C08983=1030.754,339.492,-131.948,171.836,46.140,159.013
C08984=1030.746,339.245,-131.912,171.829,46.139,159.012
C08985=1030.738,338.997,-131.876,171.824,46.139,159.011
C08986=1030.731,338.751,-131.839,171.818,46.137,159.010
C08987=1030.723,338.504,-131.803,171.812,46.137,159.009
C08988=1030.716,338.256,-131.767,171.806,46.135,159.008
C08989=1030.709,338.008,-131.730,171.800,46.135,159.007
C08990=1030.701,337.761,-131.694,171.795,46.133,159.006
C08991=1030.694,337.514,-131.658,171.789,46.133,159.006
C08992=1030.686,337.267,-131.621,171.783,46.132,159.005
C08993=1030.678,337.020,-131.585,171.778,46.131,159.004
C08994=1030.671,336.772,-131.549,171.772,46.130,159.003
C08995=1030.663,336.526,-131.513,171.766,46.129,159.002
C08996=1030.651,336.113,-131.452,171.757,46.128,159.001
C08997=1030.639,335.700,-131.391,171.748,46.126,158.999
C08998=1030.627,335.287,-131.331,171.738,46.124,158.998
C08999=1030.615,334.875,-131.271,171.729,46.123,158.996
C09000=1030.607,334.627,-131.235,171.723,46.123,158.996
C09001=1030.600,334.381,-131.199,171.718,46.121,158.995
C09002=1030.592,334.133,-131.163,171.712,46.121,158.994
C09003=1030.585,333.886,-131.128,171.707,46.120,158.993
C09004=1030.578,333.638,-131.091,171.701,46.119,158.992
C09005=1030.570,333.391,-131.055,171.695,46.119,158.991
C09006=1030.563,333.143,-131.020,171.690,46.118,158.991
C09007=1030.555,332.896,-130.984,171.684,46.117,158.990
C09008=1030.547,332.649,-130.948,171.678,46.117,158.989
C09009=1030.540,332.402,-130.913,171.673,46.116,158.988
C09010=1030.533,332.154,-130.877,171.667,46.115,158.987
C09011=1030.526,331.907,-130.841,171.662,46.114,158.987
C09012=1030.518,331.659,-130.806,171.656,46.113,158.986
C09013=1030.511,331.413,-130.770,171.651,46.113,158.985
C09014=1030.504,331.164,-130.734,171.646,46.112,158.984
C09015=1030.497,330.918,-130.698,171.640,46.111,158.983
C09016=1030.489,330.670,-130.663,171.635,46.111,158.983
C09017=1030.482,330.423,-130.628,171.629,46.111,158.982
C09018=1030.474,330.175,-130.592,171.624,46.110,158.981
C09019=1030.467,329.928,-130.556,171.619,46.109,158.980
C09020=1030.460,329.680,-130.521,171.613,46.109,158.980
C09021=1030.453,329.434,-130.485,171.608,46.108,158.979
C09022=1030.445,329.186,-130.449,171.602,46.107,158.978
C09023=1030.438,328.938,-130.415,171.597,46.106,158.977
C09024=1030.431,328.692,-130.379,171.591,46.106,158.976
C09025=1030.423,328.444,-130.343,171.586,46.105,158.976
C09026=1030.417,328.196,-130.308,171.581,46.105,158.975
C09027=1030.409,327.949,-130.272,171.576,46.104,158.974
C09028=1030.402,327.702,-130.237,171.570,46.104,158.974
C09029=1030.395,327.454,-130.202,171.565,46.103,158.973
C09030=1030.387,327.207,-130.168,171.559,46.103,158.972
C09031=1030.380,326.959,-130.132,171.554,46.102,158.971
C09032=1030.372,326.712,-130.098,171.548,46.101,158.971
C09033=1030.365,326.464,-130.062,171.543,46.101,158.970
C09034=1030.357,326.217,-130.028,171.538,46.101,158.969
C09035=1030.350,325.970,-129.992,171.532,46.101,158.969
C09036=1030.342,325.723,-129.957,171.528,46.100,158.968
C09037=1030.336,325.475,-129.923,171.522,46.100,158.967
C09038=1030.328,325.227,-129.888,171.517,46.099,158.966
C09039=1030.320,324.980,-129.853,171.511,46.098,158.966
C09040=1030.313,324.733,-129.818,171.507,46.098,158.965
C09041=1030.305,324.485,-129.783,171.501,46.098,158.964
C09042=1030.299,324.237,-129.748,171.496,46.097,158.964
C09043=1030.291,323.990,-129.714,171.490,46.097,158.963
C09044=1030.284,323.742,-129.678,171.486,46.097,158.962
C09045=1030.276,323.495,-129.643,171.480,46.097,158.962
C09046=1030.269,323.248,-129.609,171.475,46.096,158.961
C09047=1030.262,323.000,-129.575,171.469,46.096,158.960
C09048=1030.254,322.752,-129.540,171.465,46.095,158.959
C09049=1030.247,322.505,-129.504,171.459,46.095,158.959
C09050=1030.240,322.258,-129.470,171.454,46.095,158.958
C09051=1030.233,322.010,-129.436,171.449,46.094,158.957
C09052=1030.221,321.593,-129.377,171.440,46.093,158.956
C09053=1030.208,321.176,-129.319,171.432,46.093,158.955
C09054=1030.196,320.759,-129.260,171.423,46.092,158.954
C09055=1030.184,320.342,-129.203,171.415,46.092,158.953
C09056=1030.178,320.095,-129.167,171.409,46.092,158.952
C09057=1030.170,319.848,-129.133,171.404,46.091,158.952
C09058=1030.162,319.599,-129.099,171.400,46.091,158.951
C09059=1030.156,319.352,-129.064,171.394,46.091,158.950
C09060=1030.148,319.104,-129.030,171.389,46.090,158.950
C09061=1030.142,318.857,-128.995,171.384,46.090,158.949
C09062=1030.134,318.609,-128.961,171.379,46.090,158.949
C09063=1030.127,318.362,-128.926,171.374,46.089,158.948
C09064=1030.120,318.114,-128.892,171.369,46.089,158.947
C09065=1030.113,317.867,-128.857,171.364,46.089,158.947
C09066=1030.106,317.619,-128.824,171.359,46.089,158.946
C09067=1030.099,317.372,-128.788,171.354,46.089,158.945
C09068=1030.092,317.124,-128.755,171.349,46.089,158.945
C09069=1030.085,316.876,-128.720,171.344,46.089,158.944
C09070=1030.078,316.629,-128.686,171.339,46.088,158.943
C09071=1030.071,316.382,-128.652,171.334,46.088,158.943
C09072=1030.064,316.134,-128.617,171.329,46.088,158.942
C09073=1030.057,315.887,-128.583,171.324,46.087,158.942
C09074=1030.050,315.640,-128.549,171.319,46.087,158.941
C09075=1030.043,315.392,-128.514,171.315,46.087,158.940
C09076=1030.036,315.145,-128.480,171.309,46.087,158.940
C09077=1030.030,314.897,-128.446,171.304,46.087,158.939
C09078=1030.022,314.649,-128.412,171.300,46.086,158.939
C09079=1030.015,314.402,-128.378,171.294,46.086,158.938
C09080=1030.008,314.154,-128.343,171.290,46.086,158.937
C09081=1030.002,313.907,-128.310,171.285,46.086,158.937
C09082=1029.995,313.659,-128.276,171.279,46.086,158.936
C09083=1029.988,313.411,-128.241,171.275,46.086,158.936
C09084=1029.981,313.164,-128.207,171.270,46.085,158.935
C09085=1029.973,312.916,-128.173,171.266,46.085,158.934
C09086=1029.968,312.669,-128.139,171.260,46.085,158.934
C09087=1029.960,312.422,-128.105,171.255,46.085,158.933
C09088=1029.953,312.174,-128.071,171.251,46.085,158.933
C09089=1029.947,311.926,-128.037,171.246,46.085,158.932
C09090=1029.940,311.679,-128.004,171.241,46.085,158.931
C09091=1029.934,311.431,-127.969,171.236,46.084,158.931
C09092=1029.926,311.183,-127.935,171.231,46.084,158.930
C09093=1029.919,310.936,-127.901,171.227,46.084,158.930
C09094=1029.913,310.689,-127.868,171.221,46.084,158.929
C09095=1029.905,310.441,-127.835,171.217,46.084,158.929
C09096=1029.897,310.194,-127.801,171.213,46.085,158.928
C09097=1029.891,309.945,-127.768,171.207,46.085,158.928
C09098=1029.883,309.698,-127.735,171.203,46.085,158.927
C09099=1029.876,309.451,-127.701,171.198,46.085,158.927
C09100=1029.869,309.203,-127.668,171.193,46.085,158.926
C09101=1029.862,308.955,-127.634,171.188,46.085,158.926
C09102=1029.854,308.708,-127.601,171.184,46.085,158.925
C09103=1029.848,308.460,-127.568,171.179,46.085,158.925
C09104=1029.841,308.212,-127.534,171.174,46.085,158.924
C09105=1029.833,307.965,-127.501,171.169,46.086,158.924
C09106=1029.826,307.717,-127.468,171.165,46.085,158.923
C09107=1029.819,307.470,-127.435,171.160,46.086,158.923
C09108=1029.807,307.057,-127.380,171.152,46.086,158.922
C09109=1029.795,306.645,-127.324,171.145,46.086,158.921
C09110=1029.784,306.233,-127.269,171.136,46.086,158.920
C09111=1029.772,305.821,-127.214,171.128,46.087,158.919
C09112=1029.765,305.573,-127.181,171.124,46.087,158.919
C09113=1029.758,305.326,-127.147,171.119,46.087,158.918
C09114=1029.751,305.077,-127.114,171.115,46.087,158.918
C09115=1029.744,304.831,-127.081,171.110,46.087,158.917
C09116=1029.737,304.582,-127.048,171.105,46.088,158.917
C09117=1029.731,304.335,-127.015,171.100,46.088,158.916
C09118=1029.723,304.087,-126.982,171.096,46.088,158.916
C09119=1029.717,303.840,-126.949,171.092,46.088,158.915
C09120=1029.709,303.592,-126.915,171.087,46.088,158.915
C09121=1029.703,303.344,-126.883,171.082,46.089,158.914
C09122=1029.695,303.097,-126.850,171.077,46.088,158.914
C09123=1029.689,302.850,-126.817,171.073,46.089,158.913
C09124=1029.682,302.601,-126.784,171.069,46.089,158.913
C09125=1029.674,302.353,-126.751,171.064,46.089,158.912
C09126=1029.668,302.106,-126.718,171.060,46.089,158.912
C09127=1029.661,301.859,-126.685,171.054,46.090,158.911
C09128=1029.654,301.610,-126.652,171.050,46.090,158.911
C09129=1029.647,301.363,-126.620,171.045,46.090,158.911
C09130=1029.641,301.115,-126.587,171.041,46.090,158.910
C09131=1029.634,300.867,-126.554,171.037,46.091,158.910
C09132=1029.626,300.620,-126.521,171.033,46.091,158.909
C09133=1029.620,300.372,-126.488,171.028,46.091,158.909
C09134=1029.613,300.124,-126.455,171.023,46.092,158.908
C09135=1029.606,299.877,-126.423,171.018,46.092,158.908
C09136=1029.600,299.629,-126.390,171.014,46.092,158.907
C09137=1029.593,299.381,-126.357,171.009,46.092,158.907
C09138=1029.586,299.134,-126.325,171.005,46.093,158.906
C09139=1029.579,298.885,-126.292,171.001,46.093,158.906
C09140=1029.573,298.638,-126.259,170.996,46.093,158.906
C09141=1029.566,298.390,-126.226,170.992,46.094,158.905
C09142=1029.559,298.142,-126.194,170.988,46.094,158.905
C09143=1029.552,297.894,-126.161,170.983,46.094,158.904
C09144=1029.546,297.647,-126.128,170.978,46.094,158.904
C09145=1029.539,297.399,-126.096,170.973,46.095,158.903
C09146=1029.532,297.151,-126.063,170.969,46.095,158.903
C09147=1029.526,296.904,-126.030,170.965,46.096,158.903
C09148=1029.518,296.656,-125.998,170.961,46.096,158.902
C09149=1029.512,296.408,-125.965,170.956,46.096,158.902
C09150=1029.506,296.161,-125.932,170.952,46.097,158.901
C09151=1029.499,295.913,-125.900,170.948,46.097,158.901
C09152=1029.492,295.665,-125.867,170.943,46.097,158.900
C09153=1029.486,295.417,-125.834,170.939,46.097,158.900
C09154=1029.479,295.169,-125.803,170.934,46.098,158.900
C09155=1029.473,294.922,-125.770,170.930,46.098,158.899
C09156=1029.466,294.674,-125.737,170.926,46.098,158.899
C09157=1029.459,294.426,-125.705,170.921,46.099,158.898
C09158=1029.452,294.179,-125.672,170.917,46.099,158.898
C09159=1029.446,293.931,-125.640,170.913,46.099,158.897
C09160=1029.439,293.684,-125.608,170.909,46.100,158.897
C09161=1029.432,293.435,-125.575,170.904,46.101,158.897
C09162=1029.425,293.187,-125.544,170.900,46.101,158.896
C09163=1029.418,292.940,-125.512,170.895,46.102,158.896
C09164=1029.407,292.544,-125.460,170.888,46.103,158.895
C09165=1029.397,292.150,-125.409,170.882,46.103,158.895
C09166=1029.385,291.754,-125.358,170.874,46.104,158.894
C09167=1029.375,291.359,-125.307,170.868,46.105,158.894
C09168=1029.368,291.112,-125.275,170.864,46.105,158.893
C09169=1029.361,290.864,-125.243,170.860,46.106,158.893
C09170=1029.354,290.616,-125.212,170.854,46.107,158.893
C09171=1029.348,290.367,-125.179,170.850,46.107,158.892
C09172=1029.341,290.120,-125.147,170.846,46.108,158.892
C09173=1029.334,289.872,-125.116,170.842,46.109,158.891
C09174=1029.327,289.625,-125.084,170.837,46.109,158.891
C09175=1029.320,289.377,-125.052,170.833,46.109,158.891
C09176=1029.314,289.129,-125.020,170.829,46.110,158.890
C09177=1029.307,288.882,-124.988,170.825,46.111,158.890
C09178=1029.300,288.633,-124.956,170.820,46.111,158.890
C09179=1029.293,288.385,-124.925,170.816,46.112,158.889
C09180=1029.286,288.137,-124.893,170.812,46.113,158.889
C09181=1029.279,287.890,-124.861,170.808,46.113,158.889
C09182=1029.273,287.642,-124.830,170.804,46.114,158.888
C09183=1029.267,287.394,-124.798,170.799,46.114,158.888
C09184=1029.260,287.146,-124.766,170.795,46.115,158.888
C09185=1029.253,286.899,-124.734,170.791,46.116,158.887
C09186=1029.246,286.651,-124.703,170.787,46.117,158.887
C09187=1029.239,286.403,-124.671,170.783,46.117,158.887
C09188=1029.233,286.155,-124.640,170.778,46.117,158.886
C09189=1029.226,285.907,-124.608,170.774,46.118,158.886
C09190=1029.219,285.658,-124.577,170.770,46.119,158.886
C09191=1029.212,285.410,-124.545,170.766,46.120,158.885
C09192=1029.205,285.163,-124.514,170.762,46.121,158.885
C09193=1029.198,284.915,-124.482,170.757,46.121,158.885
C09194=1029.192,284.667,-124.451,170.753,46.122,158.884
C09195=1029.185,284.419,-124.419,170.749,46.123,158.884
C09196=1029.178,284.171,-124.388,170.745,46.124,158.884
C09197=1029.172,283.923,-124.357,170.741,46.124,158.883
C09198=1029.164,283.675,-124.326,170.737,46.125,158.883
C09199=1029.157,283.428,-124.294,170.733,46.126,158.883
C09200=1029.151,283.180,-124.263,170.729,46.126,158.883
C09201=1029.144,282.932,-124.231,170.725,46.127,158.882
C09202=1029.137,282.684,-124.200,170.721,46.128,158.882
C09203=1029.130,282.436,-124.169,170.717,46.128,158.882
C09204=1029.124,282.187,-124.138,170.713,46.129,158.881
C09205=1029.117,281.939,-124.106,170.709,46.130,158.881
C09206=1029.111,281.692,-124.075,170.705,46.131,158.881
C09207=1029.103,281.444,-124.044,170.701,46.132,158.881
C09208=1029.097,281.197,-124.013,170.696,46.133,158.880
C09209=1029.091,280.948,-123.982,170.692,46.133,158.880
C09210=1029.084,280.700,-123.951,170.688,46.134,158.880
C09211=1029.077,280.452,-123.920,170.684,46.135,158.879
C09212=1029.070,280.205,-123.888,170.680,46.136,158.879
C09213=1029.064,279.956,-123.857,170.676,46.137,158.879
C09214=1029.057,279.708,-123.826,170.672,46.138,158.879
C09215=1029.051,279.460,-123.795,170.668,46.139,158.878
C09216=1029.043,279.213,-123.764,170.664,46.139,158.878
C09217=1029.037,278.965,-123.733,170.660,46.140,158.878
C09218=1029.031,278.717,-123.702,170.656,46.141,158.877
C09219=1029.024,278.469,-123.670,170.652,46.142,158.877
C09220=1029.014,278.086,-123.623,170.646,46.143,158.877
C09221=1029.003,277.703,-123.574,170.640,46.144,158.876
C09222=1028.993,277.320,-123.527,170.634,46.146,158.876
C09223=1028.983,276.937,-123.479,170.628,46.147,158.876
C09224=1028.976,276.689,-123.449,170.624,46.148,158.875
C09225=1028.969,276.441,-123.418,170.619,46.149,158.875
C09226=1028.963,276.193,-123.388,170.615,46.150,158.875
C09227=1028.956,275.946,-123.357,170.611,46.151,158.874
C09228=1028.949,275.697,-123.326,170.607,46.152,158.874
C09229=1028.942,275.449,-123.295,170.603,46.153,158.874
C09230=1028.935,275.201,-123.264,170.599,46.154,158.874
C09231=1028.930,274.953,-123.234,170.596,46.154,158.874
C09232=1028.923,274.705,-123.203,170.592,46.155,158.873
C09233=1028.916,274.457,-123.173,170.588,46.156,158.873
C09234=1028.909,274.209,-123.141,170.584,46.157,158.873
C09235=1028.902,273.962,-123.111,170.580,46.158,158.873
C09236=1028.896,273.713,-123.081,170.576,46.159,158.872
C09237=1028.889,273.465,-123.049,170.572,46.160,158.872
C09238=1028.882,273.217,-123.019,170.568,46.161,158.872
C09239=1028.876,272.969,-122.989,170.564,46.162,158.872
C09240=1028.869,272.721,-122.959,170.561,46.163,158.871
C09241=1028.862,272.473,-122.927,170.557,46.164,158.871
C09242=1028.855,272.225,-122.897,170.553,46.165,158.871
C09243=1028.849,271.977,-122.867,170.549,46.166,158.871
C09244=1028.842,271.729,-122.837,170.545,46.167,158.870
C09245=1028.836,271.480,-122.806,170.540,46.168,158.870
C09246=1028.829,271.233,-122.775,170.537,46.170,158.870
C09247=1028.823,270.985,-122.745,170.534,46.170,158.870
C09248=1028.816,270.736,-122.714,170.530,46.172,158.870
C09249=1028.810,270.489,-122.684,170.526,46.173,158.870
C09250=1028.803,270.240,-122.653,170.522,46.174,158.869
C09251=1028.796,269.992,-122.623,170.518,46.175,158.869
C09252=1028.789,269.744,-122.594,170.513,46.176,158.869
C09253=1028.783,269.496,-122.563,170.511,46.177,158.869
C09254=1028.776,269.248,-122.533,170.507,46.178,158.869
C09255=1028.769,269.000,-122.503,170.503,46.179,158.868
C09256=1028.763,268.752,-122.472,170.499,46.180,158.868
C09257=1028.756,268.504,-122.442,170.495,46.181,158.868
C09258=1028.750,268.256,-122.412,170.491,46.183,158.868
C09259=1028.743,268.007,-122.382,170.487,46.184,158.867
C09260=1028.736,267.760,-122.352,170.484,46.184,158.867
C09261=1028.730,267.511,-122.321,170.480,46.185,158.867
C09262=1028.723,267.263,-122.291,170.476,46.187,158.867
C09263=1028.716,267.016,-122.261,170.472,46.188,158.867
C09264=1028.710,266.767,-122.231,170.468,46.189,158.867
C09265=1028.703,266.520,-122.201,170.465,46.190,158.867
C09266=1028.696,266.271,-122.171,170.461,46.191,158.866
C09267=1028.689,266.023,-122.140,170.457,46.192,158.866
C09268=1028.683,265.775,-122.111,170.453,46.194,158.866
C09269=1028.676,265.527,-122.081,170.449,46.195,158.866
C09270=1028.670,265.279,-122.051,170.445,46.196,158.865
C09271=1028.662,265.031,-122.021,170.442,46.197,158.865
C09272=1028.657,264.782,-121.991,170.438,46.198,158.865
C09273=1028.650,264.534,-121.961,170.434,46.199,158.865
C09274=1028.643,264.286,-121.931,170.431,46.201,158.865
C09275=1028.636,264.039,-121.901,170.427,46.202,158.865
C09276=1028.626,263.660,-121.856,170.422,46.204,158.865
C09277=1028.616,263.282,-121.811,170.416,46.205,158.864
C09278=1028.606,262.904,-121.765,170.410,46.208,158.864
C09279=1028.595,262.525,-121.720,170.404,46.210,158.864
C09280=1028.590,262.277,-121.689,170.400,46.211,158.864
C09281=1028.583,262.029,-121.660,170.397,46.212,158.864
C09282=1028.576,261.781,-121.630,170.393,46.213,158.863
C09283=1028.569,261.532,-121.601,170.390,46.215,158.863
C09284=1028.563,261.285,-121.571,170.385,46.216,158.863
C09285=1028.557,261.037,-121.540,170.382,46.217,158.863
C09286=1028.549,260.788,-121.512,170.379,46.218,158.863
C09287=1028.543,260.541,-121.482,170.375,46.220,158.863
C09288=1028.536,260.292,-121.453,170.371,46.221,158.862
C09289=1028.530,260.044,-121.423,170.367,46.223,158.862
C09290=1028.523,259.796,-121.393,170.363,46.224,158.862
C09291=1028.516,259.548,-121.365,170.360,46.225,158.862
C09292=1028.509,259.299,-121.335,170.357,46.227,158.862
C09293=1028.502,259.052,-121.306,170.353,46.228,158.862
C09294=1028.495,258.803,-121.276,170.349,46.229,158.862
C09295=1028.489,258.555,-121.247,170.345,46.231,158.862
C09296=1028.481,258.307,-121.218,170.341,46.233,158.861
C09297=1028.475,258.059,-121.189,170.339,46.234,158.861
C09298=1028.468,257.810,-121.159,170.334,46.235,158.861
C09299=1028.462,257.562,-121.130,170.331,46.237,158.861
C09300=1028.455,257.314,-121.101,170.327,46.238,158.861
C09301=1028.448,257.066,-121.072,170.323,46.239,158.861
C09302=1028.441,256.817,-121.043,170.320,46.241,158.861
C09303=1028.434,256.569,-121.013,170.316,46.242,158.861
C09304=1028.428,256.321,-120.984,170.313,46.244,158.861
C09305=1028.422,256.073,-120.954,170.309,46.245,158.860
C09306=1028.414,255.824,-120.926,170.306,46.246,158.860
C09307=1028.408,255.576,-120.897,170.302,46.248,158.860
C09308=1028.401,255.328,-120.866,170.298,46.250,158.860
C09309=1028.395,255.080,-120.837,170.294,46.251,158.860
C09310=1028.388,254.832,-120.809,170.291,46.252,158.860
C09311=1028.381,254.583,-120.780,170.288,46.254,158.860
C09312=1028.375,254.335,-120.751,170.284,46.255,158.860
C09313=1028.368,254.087,-120.722,170.280,46.257,158.860
C09314=1028.361,253.838,-120.692,170.276,46.258,158.860
C09315=1028.354,253.591,-120.663,170.273,46.259,158.860
C09316=1028.348,253.343,-120.634,170.270,46.261,158.859
C09317=1028.341,253.094,-120.605,170.266,46.263,158.859
C09318=1028.335,252.846,-120.575,170.262,46.264,158.859
C09319=1028.328,252.598,-120.547,170.259,46.266,158.859
C09320=1028.322,252.350,-120.518,170.255,46.267,158.859
C09321=1028.315,252.101,-120.489,170.252,46.268,158.859
C09322=1028.308,251.853,-120.460,170.249,46.270,158.859
C09323=1028.302,251.605,-120.430,170.245,46.271,158.859
C09324=1028.295,251.356,-120.402,170.241,46.273,158.859
C09325=1028.288,251.108,-120.373,170.238,46.275,158.859
C09326=1028.282,250.860,-120.344,170.235,46.275,158.859
C09327=1028.276,250.612,-120.315,170.231,46.277,158.858
C09328=1028.269,250.364,-120.286,170.227,46.279,158.858
C09329=1028.262,250.115,-120.257,170.224,46.280,158.858
C09330=1028.256,249.867,-120.228,170.221,46.282,158.858
C09331=1028.250,249.619,-120.199,170.217,46.283,158.858
C09332=1028.239,249.239,-120.154,170.211,46.286,158.858
C09333=1028.229,248.860,-120.110,170.206,46.288,158.858
C09334=1028.220,248.480,-120.067,170.201,46.290,158.858
C09335=1028.210,248.100,-120.022,170.196,46.292,158.858
C09336=1028.203,247.852,-119.993,170.192,46.294,158.858
C09337=1028.196,247.604,-119.965,170.188,46.296,158.858
C09338=1028.190,247.356,-119.936,170.186,46.297,158.858
C09339=1028.184,247.107,-119.907,170.182,46.299,158.857
C09340=1028.178,246.859,-119.878,170.178,46.300,158.857
C09341=1028.170,246.610,-119.850,170.175,46.302,158.857
C09342=1028.164,246.362,-119.821,170.172,46.303,158.857
C09343=1028.158,246.114,-119.792,170.168,46.305,158.857
C09344=1028.151,245.866,-119.763,170.165,46.306,158.857
C09345=1028.145,245.617,-119.735,170.161,46.308,158.857
C09346=1028.139,245.369,-119.706,170.158,46.310,158.857
C09347=1028.132,245.121,-119.677,170.155,46.311,158.857
C09348=1028.126,244.873,-119.648,170.151,46.313,158.857
C09349=1028.119,244.624,-119.620,170.147,46.314,158.857
C09350=1028.113,244.376,-119.591,170.145,46.316,158.857
C09351=1028.106,244.128,-119.562,170.141,46.317,158.857
C09352=1028.100,243.879,-119.534,170.137,46.319,158.857
C09353=1028.093,243.631,-119.505,170.134,46.320,158.857
C09354=1028.087,243.383,-119.477,170.131,46.322,158.857
C09355=1028.080,243.134,-119.448,170.127,46.324,158.856
C09356=1028.073,242.887,-119.420,170.124,46.326,158.857
C09357=1028.067,242.638,-119.391,170.121,46.327,158.857
C09358=1028.061,242.390,-119.363,170.117,46.329,158.856
C09359=1028.055,242.141,-119.334,170.114,46.331,158.856
C09360=1028.048,241.893,-119.306,170.110,46.332,158.856
C09361=1028.042,241.645,-119.278,170.107,46.334,158.856
C09362=1028.035,241.397,-119.249,170.104,46.336,158.856
C09363=1028.029,241.148,-119.221,170.100,46.338,158.856
C09364=1028.022,240.900,-119.192,170.097,46.339,158.856
C09365=1028.014,240.651,-119.164,170.094,46.341,158.856
C09366=1028.008,240.403,-119.135,170.090,46.342,158.856
C09367=1028.002,240.155,-119.108,170.086,46.344,158.856
C09368=1027.996,239.906,-119.079,170.084,46.346,158.856
C09369=1027.989,239.658,-119.051,170.080,46.348,158.856
C09370=1027.982,239.410,-119.023,170.076,46.349,158.856
C09371=1027.975,239.161,-118.995,170.074,46.351,158.856
C09372=1027.969,238.913,-118.966,170.070,46.353,158.856
C09373=1027.962,238.665,-118.939,170.066,46.355,158.856
C09374=1027.956,238.416,-118.911,170.064,46.357,158.856
C09375=1027.949,238.168,-118.883,170.060,46.358,158.856
C09376=1027.942,237.920,-118.855,170.056,46.360,158.856
C09377=1027.936,237.671,-118.826,170.054,46.362,158.856
C09378=1027.929,237.423,-118.799,170.050,46.364,158.856
C09379=1027.923,237.174,-118.771,170.046,46.365,158.856
C09380=1027.916,236.926,-118.742,170.044,46.367,158.856
C09381=1027.909,236.678,-118.715,170.040,46.369,158.856
C09382=1027.903,236.429,-118.686,170.037,46.371,158.856
C09383=1027.896,236.181,-118.659,170.034,46.373,158.856
C09384=1027.890,235.932,-118.631,170.030,46.374,158.856
C09385=1027.883,235.684,-118.603,170.027,46.377,158.856
C09386=1027.877,235.437,-118.575,170.024,46.378,158.856
C09387=1027.870,235.188,-118.547,170.020,46.380,158.856
C09388=1027.859,234.802,-118.504,170.015,46.383,158.856
C09389=1027.850,234.417,-118.461,170.010,46.386,158.856
C09390=1027.839,234.031,-118.418,170.005,46.389,158.856
C09391=1027.829,233.645,-118.374,170.000,46.392,158.856
C09392=1027.823,233.397,-118.347,169.997,46.394,158.856
C09393=1027.816,233.148,-118.319,169.993,46.395,158.856
C09394=1027.810,232.900,-118.291,169.991,46.397,158.856
C09395=1027.803,232.651,-118.263,169.987,46.399,158.856
C09396=1027.797,232.403,-118.235,169.983,46.401,158.856
C09397=1027.790,232.154,-118.208,169.981,46.403,158.856
C09398=1027.783,231.906,-118.180,169.977,46.405,158.857
C09399=1027.777,231.657,-118.152,169.973,46.407,158.856
C09400=1027.770,231.410,-118.125,169.971,46.409,158.857
C09401=1027.764,231.161,-118.097,169.967,46.410,158.856
C09402=1027.758,230.913,-118.069,169.965,46.412,158.857
C09403=1027.751,230.664,-118.041,169.961,46.414,158.857
C09404=1027.744,230.416,-118.013,169.958,46.416,158.857
C09405=1027.738,230.167,-117.985,169.955,46.418,158.857
C09406=1027.731,229.918,-117.959,169.951,46.420,158.857
C09407=1027.725,229.671,-117.932,169.948,46.422,158.857
C09408=1027.718,229.422,-117.904,169.945,46.424,158.857
C09409=1027.711,229.174,-117.876,169.942,46.426,158.857
C09410=1027.705,228.925,-117.848,169.939,46.427,158.857
C09411=1027.698,228.677,-117.821,169.935,46.430,158.857
C09412=1027.691,228.428,-117.794,169.932,46.432,158.857
C09413=1027.685,228.180,-117.766,169.929,46.434,158.857
C09414=1027.679,227.932,-117.739,169.926,46.436,158.857
C09415=1027.672,227.683,-117.711,169.923,46.438,158.857
C09416=1027.665,227.435,-117.683,169.920,46.440,158.857
C09417=1027.660,227.186,-117.657,169.916,46.442,158.857
C09418=1027.653,226.938,-117.629,169.914,46.444,158.857
C09419=1027.645,226.690,-117.602,169.910,46.446,158.857
C09420=1027.639,226.441,-117.575,169.906,46.448,158.857
C09421=1027.632,226.192,-117.547,169.904,46.450,158.858
C09422=1027.626,225.945,-117.520,169.900,46.452,158.858
C09423=1027.619,225.696,-117.493,169.898,46.454,158.858
C09424=1027.613,225.447,-117.465,169.894,46.456,158.858
C09425=1027.606,225.198,-117.438,169.891,46.458,158.858
C09426=1027.600,224.950,-117.411,169.888,46.460,158.858
C09427=1027.593,224.703,-117.384,169.884,46.462,158.858
C09428=1027.586,224.453,-117.357,169.881,46.464,158.858
C09429=1027.580,224.205,-117.329,169.879,46.466,158.858
C09430=1027.573,223.956,-117.303,169.875,46.469,158.858
C09431=1027.566,223.709,-117.275,169.873,46.471,158.858
C09432=1027.560,223.459,-117.248,169.869,46.472,158.858
C09433=1027.553,223.211,-117.221,169.865,46.475,158.858
C09434=1027.546,222.963,-117.193,169.863,46.477,158.858
C09435=1027.540,222.715,-117.167,169.859,46.479,158.859
C09436=1027.534,222.466,-117.139,169.857,46.481,158.859
C09437=1027.527,222.217,-117.112,169.853,46.483,158.859
C09438=1027.520,221.970,-117.085,169.850,46.485,158.859
C09439=1027.514,221.721,-117.058,169.847,46.487,158.859
C09440=1027.507,221.472,-117.031,169.844,46.490,158.859
C09441=1027.501,221.224,-117.005,169.841,46.492,158.859
C09442=1027.494,220.975,-116.977,169.838,46.493,158.859
C09443=1027.488,220.727,-116.950,169.834,46.496,158.859
C09444=1027.477,220.333,-116.907,169.830,46.499,158.859
C09445=1027.467,219.940,-116.864,169.825,46.502,158.859
C09446=1027.456,219.546,-116.821,169.819,46.506,158.859
C09447=1027.447,219.153,-116.779,169.815,46.509,158.860
C09448=1027.440,218.904,-116.752,169.812,46.511,158.860
C09449=1027.433,218.656,-116.725,169.809,46.513,158.860
C09450=1027.427,218.407,-116.699,169.806,46.516,158.860
C09451=1027.420,218.159,-116.671,169.802,46.518,158.860
C09452=1027.413,217.910,-116.645,169.800,46.520,158.860
C09453=1027.407,217.662,-116.618,169.796,46.522,158.860
C09454=1027.400,217.413,-116.592,169.794,46.524,158.860
C09455=1027.393,217.164,-116.565,169.791,46.527,158.861
C09456=1027.387,216.917,-116.538,169.787,46.529,158.861
C09457=1027.380,216.668,-116.511,169.785,46.531,158.861
C09458=1027.374,216.420,-116.485,169.781,46.534,158.861
C09459=1027.367,216.171,-116.459,169.779,46.536,158.861
C09460=1027.360,215.922,-116.432,169.775,46.538,158.861
C09461=1027.353,215.675,-116.405,169.772,46.540,158.861
C09462=1027.347,215.425,-116.378,169.769,46.542,158.861
C09463=1027.341,215.177,-116.352,169.766,46.545,158.861
C09464=1027.334,214.928,-116.325,169.763,46.547,158.862
C09465=1027.327,214.680,-116.298,169.760,46.549,158.862
C09466=1027.321,214.432,-116.272,169.756,46.551,158.862
C09467=1027.314,214.182,-116.245,169.754,46.554,158.862
C09468=1027.308,213.934,-116.219,169.751,46.556,158.862
C09469=1027.301,213.686,-116.192,169.748,46.558,158.862
C09470=1027.294,213.438,-116.166,169.745,46.561,158.862
C09471=1027.288,213.189,-116.139,169.742,46.563,158.862
C09472=1027.281,212.940,-116.112,169.739,46.565,158.863
C09473=1027.274,212.692,-116.086,169.735,46.567,158.863
C09474=1027.268,212.443,-116.059,169.733,46.570,158.863
C09475=1027.262,212.195,-116.033,169.730,46.572,158.863
C09476=1027.255,211.946,-116.006,169.727,46.574,158.863
C09477=1027.249,211.698,-115.980,169.724,46.576,158.863
C09478=1027.242,211.449,-115.953,169.721,46.578,158.863
C09479=1027.236,211.201,-115.927,169.718,46.581,158.863
C09480=1027.229,210.952,-115.900,169.715,46.583,158.864
C09481=1027.223,210.704,-115.874,169.712,46.586,158.864
C09482=1027.216,210.455,-115.847,169.709,46.588,158.864
C09483=1027.209,210.207,-115.821,169.706,46.590,158.864
C09484=1027.202,209.958,-115.795,169.703,46.592,158.864
C09485=1027.196,209.710,-115.768,169.700,46.595,158.864
C09486=1027.189,209.461,-115.742,169.697,46.598,158.864
C09487=1027.183,209.213,-115.716,169.695,46.600,158.865
C09488=1027.176,208.964,-115.690,169.691,46.602,158.865
C09489=1027.170,208.715,-115.663,169.689,46.605,158.865
C09490=1027.164,208.467,-115.637,169.685,46.607,158.865
C09491=1027.157,208.218,-115.611,169.682,46.609,158.865
C09492=1027.150,207.970,-115.585,169.679,46.611,158.865
C09493=1027.143,207.722,-115.558,169.676,46.614,158.865
C09494=1027.137,207.473,-115.533,169.674,46.616,158.866
C09495=1027.130,207.224,-115.506,169.670,46.619,158.866
C09496=1027.124,206.976,-115.480,169.668,46.621,158.866
C09497=1027.117,206.727,-115.454,169.665,46.624,158.866
C09498=1027.110,206.479,-115.428,169.661,46.626,158.866
C09499=1027.103,206.230,-115.402,169.659,46.628,158.866
C09500=1027.093,205.841,-115.360,169.654,46.632,158.867
C09501=1027.083,205.452,-115.320,169.650,46.636,158.867
C09502=1027.072,205.063,-115.280,169.645,46.640,158.867
C09503=1027.062,204.674,-115.239,169.640,46.644,158.867
C09504=1027.037,203.632,-115.136,169.257,46.541,158.800
C09505=1027.032,203.384,-115.112,169.252,46.544,158.800
C09506=1027.025,203.135,-115.086,169.249,46.547,158.800
C09507=1027.020,202.887,-115.062,169.245,46.551,158.800
C09508=1027.014,202.637,-115.037,169.241,46.554,158.801
C09509=1027.008,202.390,-115.013,169.237,46.557,158.801
C09510=1027.002,202.140,-114.988,169.234,46.561,158.801
C09511=1026.997,201.892,-114.964,169.229,46.564,158.801
C09512=1026.991,201.642,-114.940,169.225,46.567,158.801
C09513=1026.985,201.394,-114.915,169.222,46.570,158.802
C09514=1026.978,201.145,-114.891,169.218,46.573,158.802
C09515=1026.973,200.897,-114.866,169.214,46.577,158.802
C09516=1026.967,200.648,-114.842,169.209,46.580,158.802
C09517=1026.962,200.399,-114.817,169.206,46.583,158.803
C09518=1026.956,200.150,-114.793,169.202,46.587,158.803
C09519=1026.950,199.902,-114.768,169.198,46.590,158.803
C09520=1026.944,199.653,-114.744,169.195,46.593,158.803
C09521=1026.938,199.405,-114.720,169.191,46.597,158.804
C09522=1026.931,199.156,-114.696,169.187,46.600,158.804
C09523=1026.926,198.907,-114.672,169.182,46.603,158.804
C09524=1026.919,198.658,-114.648,169.179,46.607,158.804
C09525=1026.914,198.409,-114.624,169.175,46.610,158.804
C09526=1026.907,198.160,-114.600,169.171,46.614,158.805
C09527=1026.902,197.912,-114.575,169.167,46.617,158.805
C09528=1026.896,197.662,-114.552,169.164,46.620,158.805
C09529=1026.890,197.414,-114.528,169.160,46.624,158.805
C09530=1026.884,197.165,-114.504,169.156,46.628,158.806
C09531=1026.878,196.916,-114.480,169.152,46.631,158.806
C09532=1026.872,196.668,-114.456,169.148,46.634,158.806
C09533=1026.866,196.419,-114.432,169.145,46.638,158.806
C09534=1026.860,196.170,-114.408,169.140,46.641,158.806
C09535=1026.854,195.921,-114.384,169.137,46.644,158.807
C09536=1026.848,195.673,-114.359,169.133,46.648,158.807
C09537=1026.843,195.424,-114.336,169.129,46.651,158.807
C09538=1026.836,195.175,-114.312,169.126,46.655,158.808
C09539=1026.831,194.926,-114.288,169.122,46.658,158.808
C09540=1026.824,194.677,-114.264,169.118,46.661,158.808
C09541=1026.819,194.429,-114.240,169.115,46.665,158.808
C09542=1026.813,194.180,-114.216,169.111,46.668,158.809
C09543=1026.807,193.930,-114.192,169.107,46.672,158.809
C09544=1026.801,193.682,-114.169,169.103,46.675,158.809
C09545=1026.795,193.434,-114.145,169.099,46.678,158.809
C09546=1026.789,193.185,-114.120,169.095,46.682,158.810
C09547=1026.784,192.936,-114.097,169.092,46.685,158.810
C09548=1026.778,192.687,-114.073,169.088,46.689,158.810
C09549=1026.772,192.438,-114.049,169.084,46.693,158.810
C09550=1026.766,192.190,-114.025,169.081,46.696,158.810
C09551=1026.761,191.941,-114.002,169.077,46.699,158.811
C09552=1026.754,191.692,-113.978,169.073,46.703,158.811
C09553=1026.749,191.443,-113.954,169.070,46.706,158.811
C09554=1026.743,191.194,-113.931,169.066,46.710,158.812
C09555=1026.738,190.946,-113.906,169.062,46.713,158.812
C09556=1026.731,190.697,-113.882,169.058,46.717,158.812
C09557=1026.725,190.448,-113.859,169.054,46.720,158.812
C09558=1026.720,190.199,-113.835,169.051,46.723,158.813
C09559=1026.714,189.951,-113.811,169.047,46.727,158.813
C09560=1026.708,189.701,-113.788,169.044,46.730,158.813
C09561=1026.702,189.453,-113.764,169.040,46.734,158.813
C09562=1026.697,189.204,-113.741,169.037,46.737,158.814
C09563=1026.691,188.955,-113.717,169.033,46.741,158.814
C09564=1026.685,188.707,-113.693,169.029,46.744,158.814
C09565=1026.679,188.423,-113.666,169.025,46.748,158.814
C09566=1026.672,188.140,-113.639,169.021,46.752,158.815
C09567=1026.666,187.858,-113.612,169.017,46.756,158.815
C09568=1026.659,187.575,-113.585,169.013,46.760,158.815
C09569=1026.653,187.326,-113.562,169.009,46.763,158.816
C09570=1026.648,187.078,-113.538,169.006,46.767,158.816
C09571=1026.642,186.829,-113.515,169.002,46.770,158.816
C09572=1026.637,186.580,-113.491,168.999,46.773,158.816
C09573=1026.631,186.331,-113.468,168.995,46.777,158.817
C09574=1026.624,186.082,-113.444,168.991,46.781,158.817
C09575=1026.619,185.833,-113.420,168.988,46.784,158.817
C09576=1026.613,185.585,-113.397,168.984,46.788,158.817
C09577=1026.608,185.336,-113.374,168.980,46.791,158.818
C09578=1026.603,185.087,-113.350,168.977,46.795,158.818
C09579=1026.597,184.838,-113.326,168.973,46.798,158.818
C09580=1026.592,184.589,-113.303,168.969,46.801,158.818
C09581=1026.586,184.341,-113.279,168.966,46.805,158.819
C09582=1026.580,184.092,-113.256,168.962,46.808,158.819
C09583=1026.574,183.842,-113.232,168.959,46.812,158.819
C09584=1026.568,183.594,-113.209,168.956,46.815,158.820
C09585=1026.563,183.345,-113.185,168.952,46.818,158.820
C09586=1026.557,183.096,-113.162,168.949,46.822,158.820
C09587=1026.551,182.847,-113.139,168.945,46.825,158.820
C09588=1026.546,182.598,-113.115,168.942,46.828,158.821
C09589=1026.540,182.350,-113.093,168.938,46.832,158.821
C09590=1026.534,182.101,-113.070,168.934,46.836,158.821
C09591=1026.528,181.851,-113.046,168.931,46.840,158.822
C09592=1026.522,181.602,-113.023,168.927,46.844,158.822
C09593=1026.516,181.353,-113.001,168.924,46.847,158.822
C09594=1026.510,181.105,-112.978,168.920,46.851,158.823
C09595=1026.504,180.856,-112.955,168.917,46.855,158.823
C09596=1026.498,180.608,-112.932,168.913,46.859,158.823
C09597=1026.492,180.359,-112.909,168.909,46.863,158.824
C09598=1026.486,180.110,-112.886,168.906,46.866,158.824
C09599=1026.480,179.860,-112.863,168.902,46.870,158.824
C09600=1026.474,179.612,-112.840,168.899,46.873,158.825
C09601=1026.468,179.363,-112.817,168.895,46.877,158.825
C09602=1026.462,179.114,-112.795,168.893,46.881,158.825
C09603=1026.456,178.865,-112.773,168.888,46.884,158.825
C09604=1026.451,178.616,-112.750,168.885,46.888,158.826
C09605=1026.445,178.367,-112.727,168.882,46.892,158.826
C09606=1026.438,178.118,-112.704,168.879,46.895,158.827
C09607=1026.433,177.869,-112.681,168.875,46.899,158.827
C09608=1026.427,177.620,-112.658,168.872,46.903,158.827
C09609=1026.421,177.371,-112.635,168.868,46.906,158.827
C09610=1026.415,177.123,-112.613,168.864,46.910,158.828
C09611=1026.409,176.874,-112.590,168.861,46.914,158.828
C09612=1026.403,176.625,-112.567,168.857,46.918,158.828
C09613=1026.398,176.376,-112.544,168.854,46.922,158.829
C09614=1026.391,176.128,-112.522,168.850,46.925,158.829
C09615=1026.386,175.878,-112.500,168.847,46.929,158.829
C09616=1026.380,175.629,-112.477,168.844,46.932,158.830
C09617=1026.374,175.380,-112.454,168.840,46.936,158.830
C09618=1026.368,175.132,-112.431,168.837,46.940,158.830
C09619=1026.362,174.883,-112.408,168.833,46.944,158.831
C09620=1026.356,174.634,-112.386,168.830,46.947,158.831
C09621=1026.351,174.384,-112.363,168.826,46.951,158.831
C09622=1026.344,174.136,-112.341,168.823,46.955,158.832
C09623=1026.339,173.887,-112.318,168.819,46.959,158.832
C09624=1026.333,173.638,-112.295,168.817,46.962,158.832
C09625=1026.327,173.389,-112.273,168.813,46.966,158.833
C09626=1026.321,173.140,-112.250,168.810,46.970,158.833
C09627=1026.315,172.891,-112.228,168.806,46.973,158.833
C09628=1026.310,172.643,-112.205,168.803,46.977,158.834
C09629=1026.304,172.359,-112.180,168.799,46.982,158.834
C09630=1026.297,172.076,-112.154,168.795,46.986,158.834
C09631=1026.290,171.793,-112.128,168.791,46.990,158.835
C09632=1026.284,171.509,-112.103,168.788,46.994,158.835
C09633=1026.278,171.261,-112.080,168.784,46.998,158.836
C09634=1026.272,171.012,-112.057,168.781,47.001,158.836
C09635=1026.266,170.762,-112.035,168.778,47.005,158.836
C09636=1026.260,170.514,-112.012,168.774,47.009,158.836
C09637=1026.255,170.265,-111.989,168.771,47.013,158.837
C09638=1026.249,170.016,-111.968,168.767,47.017,158.837
C09639=1026.243,169.767,-111.945,168.764,47.020,158.838
C09640=1026.238,169.518,-111.923,168.761,47.024,158.838
C09641=1026.232,169.269,-111.900,168.757,47.027,158.838
C09642=1026.226,169.020,-111.878,168.754,47.031,158.838
C09643=1026.220,168.771,-111.855,168.751,47.035,158.839
C09644=1026.215,168.523,-111.833,168.747,47.039,158.839
C09645=1026.209,168.274,-111.811,168.745,47.042,158.840
C09646=1026.203,168.024,-111.788,168.741,47.046,158.840
C09647=1026.197,167.776,-111.765,168.737,47.049,158.840
C09648=1026.192,167.526,-111.743,168.735,47.053,158.840
C09649=1026.186,167.278,-111.721,168.731,47.057,158.841
C09650=1026.181,167.029,-111.699,168.728,47.061,158.841
C09651=1026.175,166.780,-111.676,168.725,47.065,158.842
C09652=1026.169,166.531,-111.654,168.721,47.069,158.842
C09653=1026.164,166.282,-111.632,168.718,47.072,158.842
C09654=1026.158,166.033,-111.610,168.715,47.075,158.842
C09655=1026.152,165.784,-111.587,168.711,47.079,158.843
C09656=1026.146,165.535,-111.565,168.708,47.083,158.843
C09657=1026.141,165.287,-111.542,168.705,47.087,158.844
C09658=1026.136,165.037,-111.520,168.701,47.091,158.844
C09659=1026.129,164.788,-111.498,168.699,47.094,158.844
C09660=1026.124,164.539,-111.476,168.696,47.098,158.845
C09661=1026.119,164.291,-111.453,168.692,47.101,158.845
C09662=1026.113,164.042,-111.431,168.689,47.105,158.845
C09663=1026.107,163.793,-111.408,168.686,47.109,158.846
C09664=1026.102,163.544,-111.387,168.683,47.113,158.846
C09665=1026.096,163.295,-111.365,168.679,47.117,158.846
C09666=1026.090,163.046,-111.342,168.676,47.120,158.847
C09667=1026.085,162.796,-111.320,168.673,47.124,158.847
C09668=1026.079,162.548,-111.298,168.669,47.127,158.847
C09669=1026.073,162.299,-111.275,168.666,47.131,158.847
C09670=1026.068,162.049,-111.253,168.663,47.135,158.848
C09671=1026.062,161.801,-111.231,168.660,47.139,158.848
C09672=1026.057,161.552,-111.209,168.657,47.143,158.849
C09673=1026.052,161.303,-111.187,168.654,47.146,158.849
C09674=1026.046,161.054,-111.164,168.651,47.150,158.849
C09675=1026.040,160.805,-111.143,168.648,47.153,158.850
C09676=1026.035,160.556,-111.121,168.644,47.157,158.850
C09677=1026.029,160.307,-111.098,168.641,47.161,158.850
C09678=1026.023,160.058,-111.076,168.638,47.165,158.851
C09679=1026.019,159.809,-111.054,168.635,47.168,158.851
C09680=1026.013,159.560,-111.031,168.631,47.172,158.851
C09681=1026.007,159.312,-111.010,168.628,47.176,158.852
C09682=1026.002,159.062,-110.988,168.625,47.180,158.852
C09683=1025.996,158.813,-110.966,168.623,47.183,158.852
C09684=1025.990,158.565,-110.945,168.619,47.187,158.853
C09685=1025.984,158.315,-110.923,168.616,47.191,158.853
C09686=1025.978,158.066,-110.901,168.613,47.195,158.854
C09687=1025.973,157.817,-110.880,168.609,47.199,158.854
C09688=1025.967,157.568,-110.858,168.606,47.203,158.854
C09689=1025.961,157.319,-110.837,168.603,47.206,158.855
C09690=1025.955,157.070,-110.815,168.599,47.210,158.855
C09691=1025.949,156.822,-110.792,168.597,47.214,158.855
C09692=1025.943,156.572,-110.771,168.594,47.218,158.856
C09693=1025.935,156.207,-110.739,168.588,47.224,158.856
C09694=1025.927,155.843,-110.708,168.584,47.229,158.857
C09695=1025.918,155.478,-110.676,168.580,47.235,158.857
C09696=1025.910,155.113,-110.644,168.575,47.241,158.858
C09697=1025.904,154.865,-110.623,168.572,47.245,158.858
C09698=1025.899,154.615,-110.601,168.569,47.249,158.859
C09699=1025.892,154.366,-110.579,168.566,47.253,158.859
C09700=1025.887,154.117,-110.558,168.563,47.256,158.859
C09701=1025.881,153.868,-110.536,168.559,47.260,158.860
C09702=1025.876,153.619,-110.515,168.557,47.264,158.860
C09703=1025.870,153.370,-110.494,168.554,47.268,158.861
C09704=1025.864,153.121,-110.472,168.551,47.272,158.861
C09705=1025.858,152.872,-110.451,168.547,47.276,158.861
C09706=1025.852,152.623,-110.429,168.544,47.279,158.862
C09707=1025.847,152.374,-110.408,168.541,47.284,158.862
C09708=1025.840,152.125,-110.386,168.538,47.288,158.862
C09709=1025.835,151.876,-110.366,168.535,47.292,158.863
C09710=1025.829,151.627,-110.344,168.532,47.295,158.863
C09711=1025.823,151.378,-110.323,168.529,47.299,158.864
C09712=1025.817,151.129,-110.301,168.525,47.303,158.864
C09713=1025.812,150.880,-110.280,168.523,47.307,158.864
C09714=1025.807,150.630,-110.258,168.520,47.311,158.865
C09715=1025.801,150.382,-110.237,168.517,47.315,158.865
C09716=1025.795,150.133,-110.215,168.513,47.319,158.866
C09717=1025.789,149.884,-110.194,168.510,47.323,158.866
C09718=1025.783,149.634,-110.173,168.507,47.327,158.866
C09719=1025.778,149.386,-110.152,168.504,47.330,158.867
C09720=1025.772,149.136,-110.130,168.502,47.335,158.867
C09721=1025.766,148.888,-110.109,168.498,47.339,158.868
C09722=1025.760,148.638,-110.088,168.495,47.342,158.868
C09723=1025.755,148.390,-110.067,168.492,47.346,158.868
C09724=1025.749,148.140,-110.045,168.489,47.350,158.869
C09725=1025.743,147.891,-110.025,168.485,47.354,158.869
C09726=1025.737,147.642,-110.003,168.483,47.358,158.869
C09727=1025.732,147.394,-109.982,168.480,47.362,158.870
C09728=1025.726,147.144,-109.961,168.477,47.366,158.870
C09729=1025.720,146.895,-109.940,168.474,47.370,158.871
C09730=1025.715,146.647,-109.918,168.470,47.374,158.871
C09731=1025.709,146.397,-109.897,168.468,47.377,158.871
C09732=1025.703,146.148,-109.876,168.465,47.382,158.872
C09733=1025.697,145.899,-109.855,168.462,47.386,158.872
C09734=1025.691,145.650,-109.835,168.458,47.390,158.873
C09735=1025.685,145.401,-109.814,168.455,47.393,158.873
C09736=1025.680,145.152,-109.792,168.453,47.398,158.873
C09737=1025.674,144.903,-109.772,168.450,47.402,158.874
C09738=1025.668,144.654,-109.750,168.447,47.405,158.874
C09739=1025.662,144.405,-109.730,168.443,47.409,158.874
C09740=1025.656,144.156,-109.709,168.441,47.414,158.875
C09741=1025.647,143.739,-109.674,168.436,47.420,158.876
C09742=1025.637,143.322,-109.638,168.431,47.427,158.876
C09743=1025.627,142.905,-109.604,168.426,47.434,158.877
C09744=1025.618,142.488,-109.569,168.421,47.440,158.878
C09745=1025.611,142.239,-109.548,168.418,47.445,158.878
C09746=1025.606,141.990,-109.527,168.415,47.448,158.879
C09747=1025.601,141.741,-109.506,168.412,47.452,158.879
C09748=1025.595,141.491,-109.485,168.409,47.456,158.879
C09749=1025.589,141.243,-109.465,168.406,47.461,158.880
C09750=1025.583,140.994,-109.444,168.403,47.464,158.880
C09751=1025.577,140.744,-109.423,168.400,47.468,158.881
C09752=1025.572,140.496,-109.402,168.397,47.472,158.881
C09753=1025.565,140.211,-109.378,168.394,47.477,158.881
C09754=1025.559,139.927,-109.354,168.390,47.481,158.882
C09755=1025.553,139.644,-109.331,168.387,47.486,158.882
C09756=1025.546,139.360,-109.307,168.383,47.491,158.883
C09757=1025.540,139.111,-109.287,168.380,47.495,158.883
C09758=1025.534,138.861,-109.266,168.378,47.498,158.884
C09759=1025.528,138.613,-109.244,168.375,47.502,158.884
C09760=1025.523,138.363,-109.224,168.372,47.507,158.884
C09761=1025.517,138.114,-109.204,168.369,47.510,158.885
C09762=1025.511,137.865,-109.183,168.365,47.514,158.885
C09763=1025.505,137.616,-109.163,168.363,47.519,158.886
C09764=1025.499,137.367,-109.141,168.360,47.523,158.886
C09765=1025.494,137.118,-109.121,168.357,47.526,158.886
C09766=1025.488,136.869,-109.101,168.354,47.530,158.887
C09767=1025.483,136.620,-109.080,168.352,47.535,158.887
C09768=1025.476,136.370,-109.060,168.348,47.539,158.888
C09769=1025.471,136.122,-109.039,168.345,47.542,158.888
C09770=1025.465,135.873,-109.018,168.343,47.547,158.889
C09771=1025.459,135.623,-108.998,168.340,47.551,158.889
C09772=1025.453,135.374,-108.977,168.337,47.554,158.889
C09773=1025.447,135.125,-108.957,168.334,47.559,158.890
C09774=1025.442,134.876,-108.937,168.331,47.563,158.890
C09775=1025.436,134.626,-108.916,168.328,47.567,158.891
C09776=1025.430,134.377,-108.896,168.325,47.571,158.891
C09777=1025.424,134.129,-108.875,168.322,47.575,158.891
C09778=1025.419,133.880,-108.855,168.320,47.579,158.892
C09779=1025.412,133.630,-108.834,168.317,47.583,158.892
C09780=1025.407,133.381,-108.814,168.314,47.587,158.893
C09781=1025.401,133.133,-108.794,168.311,47.592,158.893
C09782=1025.396,132.883,-108.773,168.308,47.595,158.894
C09783=1025.389,132.634,-108.753,168.305,47.599,158.894
C09784=1025.384,132.385,-108.732,168.302,47.604,158.894
C09785=1025.378,132.136,-108.712,168.299,47.607,158.895
C09786=1025.373,131.887,-108.692,168.297,47.611,158.895
C09787=1025.367,131.638,-108.672,168.294,47.615,158.896
C09788=1025.361,131.388,-108.651,168.291,47.619,158.896
C09789=1025.355,131.139,-108.631,168.287,47.624,158.896
C09790=1025.349,130.890,-108.611,168.285,47.627,158.897
C09791=1025.343,130.641,-108.591,168.282,47.632,158.897
C09792=1025.338,130.392,-108.570,168.279,47.636,158.898
C09793=1025.332,130.143,-108.550,168.276,47.639,158.898
C09794=1025.326,129.894,-108.529,168.274,47.644,158.899
C09795=1025.320,129.645,-108.509,168.271,47.648,158.899
C09796=1025.315,129.395,-108.490,168.267,47.652,158.899
C09797=1025.309,129.147,-108.470,168.265,47.656,158.900
C09798=1025.302,128.897,-108.450,168.262,47.661,158.900
C09799=1025.296,128.648,-108.430,168.259,47.664,158.901
C09800=1025.291,128.399,-108.409,168.257,47.669,158.901
C09801=1025.285,128.150,-108.390,168.254,47.673,158.902
C09802=1025.279,127.901,-108.370,168.250,47.677,158.902
C09803=1025.273,127.652,-108.350,168.247,47.681,158.902
C09804=1025.267,127.403,-108.330,168.245,47.686,158.903
C09805=1025.261,127.154,-108.309,168.242,47.689,158.903
C09806=1025.256,126.904,-108.290,168.240,47.694,158.904
C09807=1025.250,126.655,-108.270,168.237,47.698,158.904
C09808=1025.244,126.406,-108.250,168.233,47.702,158.905
C09809=1025.238,126.158,-108.230,168.230,47.706,158.905
C09810=1025.231,125.907,-108.210,168.228,47.711,158.906
C09811=1025.226,125.658,-108.190,168.225,47.715,158.906
C09812=1025.220,125.410,-108.170,168.222,47.719,158.907
C09813=1025.214,125.160,-108.151,168.220,47.723,158.907
C09814=1025.208,124.911,-108.131,168.217,47.727,158.907
C09815=1025.202,124.663,-108.111,168.213,47.731,158.908
C09816=1025.197,124.413,-108.091,168.210,47.735,158.908
C09817=1025.190,124.128,-108.068,168.208,47.740,158.909
C09818=1025.184,123.845,-108.046,168.205,47.745,158.909
C09819=1025.177,123.560,-108.023,168.201,47.750,158.910
C09820=1025.170,123.277,-108.001,168.199,47.754,158.910
C09821=1025.165,123.028,-107.980,168.195,47.758,158.911
C09822=1025.159,122.779,-107.960,168.192,47.763,158.911
C09823=1025.153,122.529,-107.941,168.189,47.767,158.912
C09824=1025.147,122.280,-107.921,168.187,47.770,158.912
C09825=1025.141,122.031,-107.901,168.184,47.775,158.912
C09826=1025.135,121.782,-107.882,168.181,47.779,158.913
C09827=1025.129,121.533,-107.862,168.179,47.783,158.913
C09828=1025.124,121.283,-107.842,168.176,47.787,158.914
C09829=1025.118,121.034,-107.822,168.173,47.792,158.914
C09830=1025.112,120.785,-107.802,168.171,47.795,158.915
C09831=1025.106,120.536,-107.783,168.168,47.799,158.915
C09832=1025.100,120.287,-107.763,168.164,47.804,158.915
C09833=1025.095,120.038,-107.743,168.161,47.808,158.916
C09834=1025.089,119.789,-107.723,168.159,47.812,158.916
C09835=1025.084,119.539,-107.704,168.156,47.816,158.917
C09836=1025.078,119.290,-107.684,168.153,47.820,158.917
C09837=1025.072,119.041,-107.664,168.151,47.824,158.918
C09838=1025.066,118.792,-107.644,168.148,47.828,158.918
C09839=1025.060,118.543,-107.625,168.145,47.833,158.919
C09840=1025.054,118.294,-107.605,168.142,47.836,158.919
C09841=1025.049,118.044,-107.585,168.140,47.840,158.919
C09842=1025.043,117.795,-107.565,168.137,47.845,158.920
C09843=1025.038,117.546,-107.546,168.134,47.849,158.920
C09844=1025.032,117.297,-107.526,168.132,47.853,158.921
C09845=1025.026,117.048,-107.507,168.129,47.857,158.921
C09846=1025.020,116.799,-107.487,168.126,47.861,158.921
C09847=1025.014,116.549,-107.468,168.124,47.865,158.922
C09848=1025.008,116.301,-107.448,168.121,47.869,158.922
C09849=1025.003,116.051,-107.428,168.118,47.873,158.923
C09850=1024.997,115.802,-107.408,168.115,47.877,158.923
C09851=1024.992,115.553,-107.389,168.113,47.881,158.924
C09852=1024.986,115.304,-107.369,168.110,47.886,158.924
C09853=1024.980,115.054,-107.350,168.107,47.889,158.925
C09854=1024.974,114.805,-107.330,168.105,47.893,158.925
C09855=1024.969,114.557,-107.311,168.102,47.898,158.925
C09856=1024.964,114.307,-107.291,168.099,47.902,158.926
C09857=1024.958,114.058,-107.271,168.096,47.905,158.926
C09858=1024.952,113.809,-107.252,168.094,47.910,158.927
C09859=1024.947,113.559,-107.232,168.091,47.914,158.927
C09860=1024.941,113.311,-107.212,168.088,47.918,158.927
C09861=1024.935,113.061,-107.193,168.086,47.922,158.928
C09862=1024.929,112.812,-107.174,168.083,47.926,158.928
C09863=1024.923,112.563,-107.154,168.080,47.930,158.929
C09864=1024.918,112.313,-107.135,168.077,47.934,158.929
C09865=1024.912,112.064,-107.116,168.074,47.938,158.930
C09866=1024.906,111.815,-107.096,168.071,47.943,158.930
C09867=1024.900,111.566,-107.076,168.068,47.947,158.930
C09868=1024.895,111.317,-107.057,168.066,47.951,158.931
C09869=1024.889,111.068,-107.039,168.063,47.955,158.931
C09870=1024.883,110.818,-107.020,168.061,47.959,158.932
C09871=1024.877,110.569,-107.000,168.058,47.963,158.932
C09872=1024.871,110.320,-106.980,168.055,47.968,158.933
C09873=1024.866,110.071,-106.961,168.052,47.972,158.933
C09874=1024.860,109.821,-106.942,168.050,47.976,158.934
C09875=1024.853,109.572,-106.923,168.047,47.980,158.934
C09876=1024.848,109.323,-106.904,168.045,47.984,158.935
C09877=1024.842,109.073,-106.885,168.042,47.988,158.935
C09878=1024.836,108.825,-106.866,168.039,47.993,158.935
C09879=1024.831,108.576,-106.847,168.037,47.997,158.936
C09880=1024.825,108.327,-106.827,168.034,48.001,158.936
C09881=1024.818,108.043,-106.806,168.030,48.006,158.937
C09882=1024.811,107.758,-106.784,168.027,48.011,158.937
C09883=1024.805,107.473,-106.763,168.025,48.016,158.938
C09884=1024.797,107.190,-106.741,168.021,48.021,158.938
C09885=1024.792,106.941,-106.722,168.018,48.025,158.939
C09886=1024.786,106.691,-106.702,168.016,48.029,158.939
C09887=1024.779,106.442,-106.684,168.013,48.033,158.940
C09888=1024.774,106.193,-106.665,168.011,48.037,158.940
C09889=1024.769,105.944,-106.646,168.008,48.041,158.941
C09890=1024.762,105.695,-106.627,168.005,48.046,158.941
C09891=1024.757,105.445,-106.608,168.003,48.050,158.941
C09892=1024.751,105.196,-106.589,168.000,48.054,158.942
C09893=1024.744,104.947,-106.570,167.997,48.058,158.942
C09894=1024.739,104.697,-106.551,167.995,48.062,158.943
C09895=1024.734,104.449,-106.532,167.991,48.067,158.943
C09896=1024.727,104.200,-106.513,167.988,48.071,158.944
C09897=1024.722,103.950,-106.494,167.986,48.075,158.944
C09898=1024.716,103.700,-106.475,167.983,48.079,158.945
C09899=1024.710,103.451,-106.457,167.980,48.083,158.945
C09900=1024.705,103.202,-106.438,167.978,48.088,158.945
C09901=1024.699,102.953,-106.419,167.975,48.092,158.946
C09902=1024.693,102.704,-106.400,167.973,48.096,158.946
C09903=1024.687,102.454,-106.381,167.970,48.100,158.947
C09904=1024.682,102.206,-106.362,167.967,48.105,158.947
C09905=1024.675,101.956,-106.343,167.964,48.108,158.948
C09906=1024.670,101.707,-106.324,167.962,48.113,158.948
C09907=1024.663,101.458,-106.305,167.959,48.117,158.949
C09908=1024.658,101.209,-106.286,167.957,48.121,158.949
C09909=1024.653,100.959,-106.268,167.954,48.125,158.949
C09910=1024.646,100.710,-106.249,167.951,48.129,158.950
C09911=1024.641,100.461,-106.230,167.949,48.134,158.950
C09912=1024.636,100.212,-106.211,167.946,48.137,158.951
C09913=1024.629,99.963,-106.192,167.943,48.142,158.951
C09914=1024.623,99.713,-106.173,167.940,48.146,158.952
C09915=1024.618,99.463,-106.155,167.938,48.150,158.952
C09916=1024.612,99.215,-106.136,167.935,48.154,158.952
C09917=1024.606,98.966,-106.118,167.933,48.159,158.953
C09918=1024.600,98.716,-106.099,167.930,48.163,158.954
C09919=1024.594,98.466,-106.081,167.927,48.167,158.954
C09920=1024.588,98.218,-106.062,167.925,48.172,158.954
C09921=1024.582,97.969,-106.043,167.922,48.175,158.955
C09922=1024.576,97.719,-106.025,167.920,48.180,158.955
C09923=1024.570,97.470,-106.006,167.917,48.184,158.956
C09924=1024.565,97.221,-105.988,167.914,48.188,158.956
C09925=1024.559,96.971,-105.970,167.912,48.193,158.957
C09926=1024.553,96.722,-105.950,167.909,48.197,158.957
C09927=1024.547,96.473,-105.932,167.907,48.201,158.958
C09928=1024.541,96.224,-105.914,167.904,48.205,158.958
C09929=1024.535,95.974,-105.895,167.901,48.210,158.959
C09930=1024.529,95.725,-105.876,167.899,48.214,158.959
C09931=1024.523,95.476,-105.859,167.896,48.218,158.959
C09932=1024.518,95.227,-105.839,167.894,48.223,158.960
C09933=1024.512,94.977,-105.822,167.891,48.226,158.960
C09934=1024.506,94.729,-105.803,167.888,48.231,158.961
C09935=1024.500,94.479,-105.784,167.886,48.235,158.961
C09936=1024.494,94.229,-105.766,167.883,48.239,158.962
C09937=1024.488,93.981,-105.748,167.880,48.243,158.962
C09938=1024.483,93.731,-105.729,167.878,48.248,158.963
C09939=1024.476,93.482,-105.711,167.875,48.252,158.963
C09940=1024.471,93.233,-105.692,167.872,48.256,158.964
C09941=1024.465,92.983,-105.674,167.870,48.260,158.964
C09942=1024.459,92.734,-105.655,167.867,48.265,158.964
C09943=1024.453,92.485,-105.638,167.864,48.268,158.965
C09944=1024.448,92.236,-105.618,167.862,48.273,158.965
C09945=1024.441,91.951,-105.598,167.858,48.278,158.966
C09946=1024.434,91.667,-105.577,167.856,48.282,158.966
C09947=1024.428,91.384,-105.556,167.852,48.287,158.967
C09948=1024.421,91.100,-105.535,167.850,48.292,158.967
C09949=1024.415,90.850,-105.517,167.848,48.296,158.968
C09950=1024.409,90.600,-105.498,167.845,48.300,158.968
C09951=1024.404,90.351,-105.480,167.842,48.305,158.969
C09952=1024.398,90.102,-105.461,167.840,48.309,158.969
C09953=1024.393,89.853,-105.443,167.837,48.313,158.970
C09954=1024.386,89.604,-105.425,167.834,48.317,158.970
C09955=1024.380,89.354,-105.407,167.832,48.322,158.970
C09956=1024.375,89.105,-105.389,167.829,48.325,158.971
C09957=1024.368,88.856,-105.370,167.827,48.330,158.971
C09958=1024.363,88.607,-105.353,167.824,48.335,158.972
C09959=1024.357,88.357,-105.335,167.820,48.339,158.972
C09960=1024.351,88.108,-105.316,167.818,48.343,158.973
C09961=1024.345,87.859,-105.298,167.815,48.348,158.973
C09962=1024.339,87.609,-105.280,167.813,48.352,158.974
C09963=1024.333,87.360,-105.262,167.810,48.356,158.974
C09964=1024.327,87.111,-105.244,167.807,48.360,158.974
C09965=1024.321,86.861,-105.226,167.805,48.365,158.975
C09966=1024.316,86.612,-105.208,167.802,48.369,158.975
C09967=1024.309,86.363,-105.190,167.800,48.373,158.976
C09968=1024.304,86.114,-105.172,167.797,48.378,158.976
C09969=1024.298,85.864,-105.154,167.794,48.382,158.977
C09970=1024.292,85.616,-105.136,167.792,48.386,158.977
C09971=1024.286,85.366,-105.118,167.789,48.391,158.978
C09972=1024.280,85.116,-105.100,167.787,48.395,158.978
C09973=1024.274,84.867,-105.083,167.784,48.399,158.979
C09974=1024.268,84.617,-105.065,167.781,48.403,158.979
C09975=1024.262,84.369,-105.046,167.779,48.408,158.980
C09976=1024.256,84.119,-105.028,167.776,48.411,158.980
C09977=1024.250,83.870,-105.011,167.774,48.416,158.980
C09978=1024.244,83.620,-104.993,167.771,48.421,158.981
C09979=1024.239,83.372,-104.975,167.768,48.424,158.981
C09980=1024.232,83.122,-104.957,167.766,48.429,158.982
C09981=1024.227,82.873,-104.939,167.763,48.433,158.982
C09982=1024.221,82.623,-104.921,167.761,48.437,158.983
C09983=1024.215,82.374,-104.904,167.758,48.441,158.983
C09984=1024.209,82.125,-104.886,167.755,48.446,158.984
C09985=1024.203,81.876,-104.867,167.753,48.450,158.984
C09986=1024.197,81.627,-104.850,167.750,48.454,158.984
C09987=1024.192,81.377,-104.832,167.747,48.458,158.985
C09988=1024.186,81.128,-104.814,167.745,48.463,158.985
C09989=1024.180,80.879,-104.796,167.742,48.467,158.986
C09990=1024.174,80.629,-104.779,167.740,48.471,158.986
C09991=1024.168,80.380,-104.761,167.737,48.476,158.987
C09992=1024.162,80.131,-104.742,167.735,48.480,158.987
C09993=1024.156,79.882,-104.725,167.732,48.484,158.988
C09994=1024.150,79.632,-104.707,167.729,48.488,158.988
C09995=1024.145,79.383,-104.689,167.727,48.493,158.989
C09996=1024.139,79.134,-104.672,167.724,48.497,158.989
//INST
///DATE 2021/06/17 10:58
///ATTR SC,RW,RJ
////FRAME ROBOT
///GROUP1 RB1
NOP
MOVL C00000 V=800.0 PL=0
MOVL C00001 V=800.0 PL=0
MOVL C00002 V=800.0 PL=0
MOVL C00003 V=800.0 PL=0
MOVL C00004 V=800.0 PL=0
MOVL C00005 V=800.0 PL=0
MOVL C00006 V=800.0 PL=0
MOVL C00007 V=800.0 PL=0
MOVL C00008 V=800.0 PL=0
MOVL C00009 V=800.0 PL=0
MOVL C00010 V=800.0 PL=0
MOVL C00011 V=800.0 PL=0
MOVL C00012 V=800.0 PL=0
MOVL C00013 V=800.0 PL=0
MOVL C00014 V=800.0 PL=0
MOVL C00015 V=800.0 PL=0
MOVL C00016 V=800.0 PL=0
MOVL C00017 V=800.0 PL=0
MOVL C00018 V=800.0 PL=0
MOVL C00019 V=800.0 PL=0
MOVL C00020 V=800.0 PL=0
MOVL C00021 V=800.0 PL=0
MOVL C00022 V=800.0 PL=0
MOVL C00023 V=800.0 PL=0
MOVL C00024 V=800.0 PL=0
MOVL C00025 V=800.0 PL=0
MOVL C00026 V=800.0 PL=0
MOVL C00027 V=800.0 PL=0
MOVL C00028 V=800.0 PL=0
MOVL C00029 V=800.0 PL=0
MOVL C00030 V=800.0 PL=0
MOVL C00031 V=800.0 PL=0
MOVL C00032 V=800.0 PL=0
MOVL C00033 V=800.0 PL=0
MOVL C00034 V=800.0 PL=0
MOVL C00035 V=800.0 PL=0
MOVL C00036 V=800.0 PL=0
MOVL C00037 V=800.0 PL=0
MOVL C00038 V=800.0 PL=0
MOVL C00039 V=800.0 PL=0
MOVL C00040 V=800.0 PL=0
MOVL C00041 V=800.0 PL=0
MOVL C00042 V=800.0 PL=0
MOVL C00043 V=800.0 PL=0
MOVL C00044 V=800.0 PL=0
MOVL C00045 V=800.0 PL=0
MOVL C00046 V=800.0 PL=0
MOVL C00047 V=800.0 PL=0
MOVL C00048 V=800.0 PL=0
MOVL C00049 V=800.0 PL=0
MOVL C00050 V=800.0 PL=0
MOVL C00051 V=800.0 PL=0
MOVL C00052 V=800.0 PL=0
MOVL C00053 V=800.0 PL=0
MOVL C00054 V=800.0 PL=0
MOVL C00055 V=800.0 PL=0
MOVL C00056 V=800.0 PL=0
MOVL C00057 V=800.0 PL=0
MOVL C00058 V=800.0 PL=0
MOVL C00059 V=800.0 PL=0
MOVL C00060 V=800.0 PL=0
MOVL C00061 V=800.0 PL=0
MOVL C00062 V=800.0 PL=0
MOVL C00063 V=800.0 PL=0
MOVL C00064 V=800.0 PL=0
MOVL C00065 V=800.0 PL=0
MOVL C00066 V=800.0 PL=0
MOVL C00067 V=800.0 PL=0
MOVL C00068 V=800.0 PL=0
MOVL C00069 V=800.0 PL=0
MOVL C00070 V=800.0 PL=0
MOVL C00071 V=800.0 PL=0
MOVL C00072 V=800.0 PL=0
MOVL C00073 V=800.0 PL=0
MOVL C00074 V=800.0 PL=0
MOVL C00075 V=800.0 PL=0
MOVL C00076 V=800.0 PL=0
MOVL C00077 V=800.0 PL=0
MOVL C00078 V=800.0 PL=0
MOVL C00079 V=800.0 PL=0
MOVL C00080 V=800.0 PL=0
MOVL C00081 V=800.0 PL=0
MOVL C00082 V=800.0 PL=0
MOVL C00083 V=800.0 PL=0
MOVL C00084 V=800.0 PL=0
MOVL C00085 V=800.0 PL=0
MOVL C00086 V=800.0 PL=0
MOVL C00087 V=800.0 PL=0
MOVL C00088 V=800.0 PL=0
MOVL C00089 V=800.0 PL=0
MOVL C00090 V=800.0 PL=0
MOVL C00091 V=800.0 PL=0
MOVL C00092 V=800.0 PL=0
MOVL C00093 V=800.0 PL=0
MOVL C00094 V=800.0 PL=0
MOVL C00095 V=800.0 PL=0
MOVL C00096 V=800.0 PL=0
MOVL C00097 V=800.0 PL=0
MOVL C00098 V=800.0 PL=0
MOVL C00099 V=800.0 PL=0
MOVL C00100 V=800.0 PL=0
MOVL C00101 V=800.0 PL=0
MOVL C00102 V=800.0 PL=0
MOVL C00103 V=800.0 PL=0
MOVL C00104 V=800.0 PL=0
MOVL C00105 V=800.0 PL=0
MOVL C00106 V=800.0 PL=0
MOVL C00107 V=800.0 PL=0
MOVL C00108 V=800.0 PL=0
MOVL C00109 V=800.0 PL=0
MOVL C00110 V=800.0 PL=0
MOVL C00111 V=800.0 PL=0
MOVL C00112 V=800.0 PL=0
MOVL C00113 V=800.0 PL=0
MOVL C00114 V=800.0 PL=0
MOVL C00115 V=800.0 PL=0
MOVL C00116 V=800.0 PL=0
MOVL C00117 V=800.0 PL=0
MOVL C00118 V=800.0 PL=0
MOVL C00119 V=800.0 PL=0
MOVL C00120 V=800.0 PL=0
MOVL C00121 V=800.0 PL=0
MOVL C00122 V=800.0 PL=0
MOVL C00123 V=800.0 PL=0
MOVL C00124 V=800.0 PL=0
MOVL C00125 V=800.0 PL=0
MOVL C00126 V=800.0 PL=0
MOVL C00127 V=800.0 PL=0
MOVL C00128 V=800.0 PL=0
MOVL C00129 V=800.0 PL=0
MOVL C00130 V=800.0 PL=0
MOVL C00131 V=800.0 PL=0
MOVL C00132 V=800.0 PL=0
MOVL C00133 V=800.0 PL=0
MOVL C00134 V=800.0 PL=0
MOVL C00135 V=800.0 PL=0
MOVL C00136 V=800.0 PL=0
MOVL C00137 V=800.0 PL=0
MOVL C00138 V=800.0 PL=0
MOVL C00139 V=800.0 PL=0
MOVL C00140 V=800.0 PL=0
MOVL C00141 V=800.0 PL=0
MOVL C00142 V=800.0 PL=0
MOVL C00143 V=800.0 PL=0
MOVL C00144 V=800.0 PL=0
MOVL C00145 V=800.0 PL=0
MOVL C00146 V=800.0 PL=0
MOVL C00147 V=800.0 PL=0
MOVL C00148 V=800.0 PL=0
MOVL C00149 V=800.0 PL=0
MOVL C00150 V=800.0 PL=0
MOVL C00151 V=800.0 PL=0
MOVL C00152 V=800.0 PL=0
MOVL C00153 V=800.0 PL=0
MOVL C00154 V=800.0 PL=0
MOVL C00155 V=800.0 PL=0
MOVL C00156 V=800.0 PL=0
MOVL C00157 V=800.0 PL=0
MOVL C00158 V=800.0 PL=0
MOVL C00159 V=800.0 PL=0
MOVL C00160 V=800.0 PL=0
MOVL C00161 V=800.0 PL=0
MOVL C00162 V=800.0 PL=0
MOVL C00163 V=800.0 PL=0
MOVL C00164 V=800.0 PL=0
MOVL C00165 V=800.0 PL=0
MOVL C00166 V=800.0 PL=0
MOVL C00167 V=800.0 PL=0
MOVL C00168 V=800.0 PL=0
MOVL C00169 V=800.0 PL=0
MOVL C00170 V=800.0 PL=0
MOVL C00171 V=800.0 PL=0
MOVL C00172 V=800.0 PL=0
MOVL C00173 V=800.0 PL=0
MOVL C00174 V=800.0 PL=0
MOVL C00175 V=800.0 PL=0
MOVL C00176 V=800.0 PL=0
MOVL C00177 V=800.0 PL=0
MOVL C00178 V=800.0 PL=0
MOVL C00179 V=800.0 PL=0
MOVL C00180 V=800.0 PL=0
MOVL C00181 V=800.0 PL=0
MOVL C00182 V=800.0 PL=0
MOVL C00183 V=800.0 PL=0
MOVL C00184 V=800.0 PL=0
MOVL C00185 V=800.0 PL=0
MOVL C00186 V=800.0 PL=0
MOVL C00187 V=800.0 PL=0
MOVL C00188 V=800.0 PL=0
MOVL C00189 V=800.0 PL=0
MOVL C00190 V=800.0 PL=0
MOVL C00191 V=800.0 PL=0
MOVL C00192 V=800.0 PL=0
MOVL C00193 V=800.0 PL=0
MOVL C00194 V=800.0 PL=0
MOVL C00195 V=800.0 PL=0
MOVL C00196 V=800.0 PL=0
MOVL C00197 V=800.0 PL=0
MOVL C00198 V=800.0 PL=0
MOVL C00199 V=800.0 PL=0
MOVL C00200 V=800.0 PL=0
MOVL C00201 V=800.0 PL=0
MOVL C00202 V=800.0 PL=0
MOVL C00203 V=800.0 PL=0
MOVL C00204 V=800.0 PL=0
MOVL C00205 V=800.0 PL=0
MOVL C00206 V=800.0 PL=0
MOVL C00207 V=800.0 PL=0
MOVL C00208 V=800.0 PL=0
MOVL C00209 V=800.0 PL=0
MOVL C00210 V=800.0 PL=0
MOVL C00211 V=800.0 PL=0
MOVL C00212 V=800.0 PL=0
MOVL C00213 V=800.0 PL=0
MOVL C00214 V=800.0 PL=0
MOVL C00215 V=800.0 PL=0
MOVL C00216 V=800.0 PL=0
MOVL C00217 V=800.0 PL=0
MOVL C00218 V=800.0 PL=0
MOVL C00219 V=800.0 PL=0
MOVL C00220 V=800.0 PL=0
MOVL C00221 V=800.0 PL=0
MOVL C00222 V=800.0 PL=0
MOVL C00223 V=800.0 PL=0
MOVL C00224 V=800.0 PL=0
MOVL C00225 V=800.0 PL=0
MOVL C00226 V=800.0 PL=0
MOVL C00227 V=800.0 PL=0
MOVL C00228 V=800.0 PL=0
MOVL C00229 V=800.0 PL=0
MOVL C00230 V=800.0 PL=0
MOVL C00231 V=800.0 PL=0
MOVL C00232 V=800.0 PL=0
MOVL C00233 V=800.0 PL=0
MOVL C00234 V=800.0 PL=0
MOVL C00235 V=800.0 PL=0
MOVL C00236 V=800.0 PL=0
MOVL C00237 V=800.0 PL=0
MOVL C00238 V=800.0 PL=0
MOVL C00239 V=800.0 PL=0
MOVL C00240 V=800.0 PL=0
MOVL C00241 V=800.0 PL=0
MOVL C00242 V=800.0 PL=0
MOVL C00243 V=800.0 PL=0
MOVL C00244 V=800.0 PL=0
MOVL C00245 V=800.0 PL=0
MOVL C00246 V=800.0 PL=0
MOVL C00247 V=800.0 PL=0
MOVL C00248 V=800.0 PL=0
MOVL C00249 V=800.0 PL=0
MOVL C00250 V=800.0 PL=0
MOVL C00251 V=800.0 PL=0
MOVL C00252 V=800.0 PL=0
MOVL C00253 V=800.0 PL=0
MOVL C00254 V=800.0 PL=0
MOVL C00255 V=800.0 PL=0
MOVL C00256 V=800.0 PL=0
MOVL C00257 V=800.0 PL=0
MOVL C00258 V=800.0 PL=0
MOVL C00259 V=800.0 PL=0
MOVL C00260 V=800.0 PL=0
MOVL C00261 V=800.0 PL=0
MOVL C00262 V=800.0 PL=0
MOVL C00263 V=800.0 PL=0
MOVL C00264 V=800.0 PL=0
MOVL C00265 V=800.0 PL=0
MOVL C00266 V=800.0 PL=0
MOVL C00267 V=800.0 PL=0
MOVL C00268 V=800.0 PL=0
MOVL C00269 V=800.0 PL=0
MOVL C00270 V=800.0 PL=0
MOVL C00271 V=800.0 PL=0
MOVL C00272 V=800.0 PL=0
MOVL C00273 V=800.0 PL=0
MOVL C00274 V=800.0 PL=0
MOVL C00275 V=800.0 PL=0
MOVL C00276 V=800.0 PL=0
MOVL C00277 V=800.0 PL=0
MOVL C00278 V=800.0 PL=0
MOVL C00279 V=800.0 PL=0
MOVL C00280 V=800.0 PL=0
MOVL C00281 V=800.0 PL=0
MOVL C00282 V=800.0 PL=0
MOVL C00283 V=800.0 PL=0
MOVL C00284 V=800.0 PL=0
MOVL C00285 V=800.0 PL=0
MOVL C00286 V=800.0 PL=0
MOVL C00287 V=800.0 PL=0
MOVL C00288 V=800.0 PL=0
MOVL C00289 V=800.0 PL=0
MOVL C00290 V=800.0 PL=0
MOVL C00291 V=800.0 PL=0
MOVL C00292 V=800.0 PL=0
MOVL C00293 V=800.0 PL=0
MOVL C00294 V=800.0 PL=0
MOVL C00295 V=800.0 PL=0
MOVL C00296 V=800.0 PL=0
MOVL C00297 V=800.0 PL=0
MOVL C00298 V=800.0 PL=0
MOVL C00299 V=800.0 PL=0
MOVL C00300 V=800.0 PL=0
MOVL C00301 V=800.0 PL=0
MOVL C00302 V=800.0 PL=0
MOVL C00303 V=800.0 PL=0
MOVL C00304 V=800.0 PL=0
MOVL C00305 V=800.0 PL=0
MOVL C00306 V=800.0 PL=0
MOVL C00307 V=800.0 PL=0
MOVL C00308 V=800.0 PL=0
MOVL C00309 V=800.0 PL=0
MOVL C00310 V=800.0 PL=0
MOVL C00311 V=800.0 PL=0
MOVL C00312 V=800.0 PL=0
MOVL C00313 V=800.0 PL=0
MOVL C00314 V=800.0 PL=0
MOVL C00315 V=800.0 PL=0
MOVL C00316 V=800.0 PL=0
MOVL C00317 V=800.0 PL=0
MOVL C00318 V=800.0 PL=0
MOVL C00319 V=800.0 PL=0
MOVL C00320 V=800.0 PL=0
MOVL C00321 V=800.0 PL=0
MOVL C00322 V=800.0 PL=0
MOVL C00323 V=800.0 PL=0
MOVL C00324 V=800.0 PL=0
MOVL C00325 V=800.0 PL=0
MOVL C00326 V=800.0 PL=0
MOVL C00327 V=800.0 PL=0
MOVL C00328 V=800.0 PL=0
MOVL C00329 V=800.0 PL=0
MOVL C00330 V=800.0 PL=0
MOVL C00331 V=800.0 PL=0
MOVL C00332 V=800.0 PL=0
MOVL C00333 V=800.0 PL=0
MOVL C00334 V=800.0 PL=0
MOVL C00335 V=800.0 PL=0
MOVL C00336 V=800.0 PL=0
MOVL C00337 V=800.0 PL=0
MOVL C00338 V=800.0 PL=0
MOVL C00339 V=800.0 PL=0
MOVL C00340 V=800.0 PL=0
MOVL C00341 V=800.0 PL=0
MOVL C00342 V=800.0 PL=0
MOVL C00343 V=800.0 PL=0
MOVL C00344 V=800.0 PL=0
MOVL C00345 V=800.0 PL=0
MOVL C00346 V=800.0 PL=0
MOVL C00347 V=800.0 PL=0
MOVL C00348 V=800.0 PL=0
MOVL C00349 V=800.0 PL=0
MOVL C00350 V=800.0 PL=0
MOVL C00351 V=800.0 PL=0
MOVL C00352 V=800.0 PL=0
MOVL C00353 V=800.0 PL=0
MOVL C00354 V=800.0 PL=0
MOVL C00355 V=800.0 PL=0
MOVL C00356 V=800.0 PL=0
MOVL C00357 V=800.0 PL=0
MOVL C00358 V=800.0 PL=0
MOVL C00359 V=800.0 PL=0
MOVL C00360 V=800.0 PL=0
MOVL C00361 V=800.0 PL=0
MOVL C00362 V=800.0 PL=0
MOVL C00363 V=800.0 PL=0
MOVL C00364 V=800.0 PL=0
MOVL C00365 V=800.0 PL=0
MOVL C00366 V=800.0 PL=0
MOVL C00367 V=800.0 PL=0
MOVL C00368 V=800.0 PL=0
MOVL C00369 V=800.0 PL=0
MOVL C00370 V=800.0 PL=0
MOVL C00371 V=800.0 PL=0
MOVL C00372 V=800.0 PL=0
MOVL C00373 V=800.0 PL=0
MOVL C00374 V=800.0 PL=0
MOVL C00375 V=800.0 PL=0
MOVL C00376 V=800.0 PL=0
MOVL C00377 V=800.0 PL=0
MOVL C00378 V=800.0 PL=0
MOVL C00379 V=800.0 PL=0
MOVL C00380 V=800.0 PL=0
MOVL C00381 V=800.0 PL=0
MOVL C00382 V=800.0 PL=0
MOVL C00383 V=800.0 PL=0
MOVL C00384 V=800.0 PL=0
MOVL C00385 V=800.0 PL=0
MOVL C00386 V=800.0 PL=0
MOVL C00387 V=800.0 PL=0
MOVL C00388 V=800.0 PL=0
MOVL C00389 V=800.0 PL=0
MOVL C00390 V=800.0 PL=0
MOVL C00391 V=800.0 PL=0
MOVL C00392 V=800.0 PL=0
MOVL C00393 V=800.0 PL=0
MOVL C00394 V=800.0 PL=0
MOVL C00395 V=800.0 PL=0
MOVL C00396 V=800.0 PL=0
MOVL C00397 V=800.0 PL=0
MOVL C00398 V=800.0 PL=0
MOVL C00399 V=800.0 PL=0
MOVL C00400 V=800.0 PL=0
MOVL C00401 V=800.0 PL=0
MOVL C00402 V=800.0 PL=0
MOVL C00403 V=800.0 PL=0
MOVL C00404 V=800.0 PL=0
MOVL C00405 V=800.0 PL=0
MOVL C00406 V=800.0 PL=0
MOVL C00407 V=800.0 PL=0
MOVL C00408 V=800.0 PL=0
MOVL C00409 V=800.0 PL=0
MOVL C00410 V=800.0 PL=0
MOVL C00411 V=800.0 PL=0
MOVL C00412 V=800.0 PL=0
MOVL C00413 V=800.0 PL=0
MOVL C00414 V=800.0 PL=0
MOVL C00415 V=800.0 PL=0
MOVL C00416 V=800.0 PL=0
MOVL C00417 V=800.0 PL=0
MOVL C00418 V=800.0 PL=0
MOVL C00419 V=800.0 PL=0
MOVL C00420 V=800.0 PL=0
MOVL C00421 V=800.0 PL=0
MOVL C00422 V=800.0 PL=0
MOVL C00423 V=800.0 PL=0
MOVL C00424 V=800.0 PL=0
MOVL C00425 V=800.0 PL=0
MOVL C00426 V=800.0 PL=0
MOVL C00427 V=800.0 PL=0
MOVL C00428 V=800.0 PL=0
MOVL C00429 V=800.0 PL=0
MOVL C00430 V=800.0 PL=0
MOVL C00431 V=800.0 PL=0
MOVL C00432 V=800.0 PL=0
MOVL C00433 V=800.0 PL=0
MOVL C00434 V=800.0 PL=0
MOVL C00435 V=800.0 PL=0
MOVL C00436 V=800.0 PL=0
MOVL C00437 V=800.0 PL=0
MOVL C00438 V=800.0 PL=0
MOVL C00439 V=800.0 PL=0
MOVL C00440 V=800.0 PL=0
MOVL C00441 V=800.0 PL=0
MOVL C00442 V=800.0 PL=0
MOVL C00443 V=800.0 PL=0
MOVL C00444 V=800.0 PL=0
MOVL C00445 V=800.0 PL=0
MOVL C00446 V=800.0 PL=0
MOVL C00447 V=800.0 PL=0
MOVL C00448 V=800.0 PL=0
MOVL C00449 V=800.0 PL=0
MOVL C00450 V=800.0 PL=0
MOVL C00451 V=800.0 PL=0
MOVL C00452 V=800.0 PL=0
MOVL C00453 V=800.0 PL=0
MOVL C00454 V=800.0 PL=0
MOVL C00455 V=800.0 PL=0
MOVL C00456 V=800.0 PL=0
MOVL C00457 V=800.0 PL=0
MOVL C00458 V=800.0 PL=0
MOVL C00459 V=800.0 PL=0
MOVL C00460 V=800.0 PL=0
MOVL C00461 V=800.0 PL=0
MOVL C00462 V=800.0 PL=0
MOVL C00463 V=800.0 PL=0
MOVL C00464 V=800.0 PL=0
MOVL C00465 V=800.0 PL=0
MOVL C00466 V=800.0 PL=0
MOVL C00467 V=800.0 PL=0
MOVL C00468 V=800.0 PL=0
MOVL C00469 V=800.0 PL=0
MOVL C00470 V=800.0 PL=0
MOVL C00471 V=800.0 PL=0
MOVL C00472 V=800.0 PL=0
MOVL C00473 V=800.0 PL=0
MOVL C00474 V=800.0 PL=0
MOVL C00475 V=800.0 PL=0
MOVL C00476 V=800.0 PL=0
MOVL C00477 V=800.0 PL=0
MOVL C00478 V=800.0 PL=0
MOVL C00479 V=800.0 PL=0
MOVL C00480 V=800.0 PL=0
MOVL C00481 V=800.0 PL=0
MOVL C00482 V=800.0 PL=0
MOVL C00483 V=800.0 PL=0
MOVL C00484 V=800.0 PL=0
MOVL C00485 V=800.0 PL=0
MOVL C00486 V=800.0 PL=0
MOVL C00487 V=800.0 PL=0
MOVL C00488 V=800.0 PL=0
MOVL C00489 V=800.0 PL=0
MOVL C00490 V=800.0 PL=0
MOVL C00491 V=800.0 PL=0
MOVL C00492 V=800.0 PL=0
MOVL C00493 V=800.0 PL=0
MOVL C00494 V=800.0 PL=0
MOVL C00495 V=800.0 PL=0
MOVL C00496 V=800.0 PL=0
MOVL C00497 V=800.0 PL=0
MOVL C00498 V=800.0 PL=0
MOVL C00499 V=800.0 PL=0
MOVL C00500 V=800.0 PL=0
MOVL C00501 V=800.0 PL=0
MOVL C00502 V=800.0 PL=0
MOVL C00503 V=800.0 PL=0
MOVL C00504 V=800.0 PL=0
MOVL C00505 V=800.0 PL=0
MOVL C00506 V=800.0 PL=0
MOVL C00507 V=800.0 PL=0
MOVL C00508 V=800.0 PL=0
MOVL C00509 V=800.0 PL=0
MOVL C00510 V=800.0 PL=0
MOVL C00511 V=800.0 PL=0
MOVL C00512 V=800.0 PL=0
MOVL C00513 V=800.0 PL=0
MOVL C00514 V=800.0 PL=0
MOVL C00515 V=800.0 PL=0
MOVL C00516 V=800.0 PL=0
MOVL C00517 V=800.0 PL=0
MOVL C00518 V=800.0 PL=0
MOVL C00519 V=800.0 PL=0
MOVL C00520 V=800.0 PL=0
MOVL C00521 V=800.0 PL=0
MOVL C00522 V=800.0 PL=0
MOVL C00523 V=800.0 PL=0
MOVL C00524 V=800.0 PL=0
MOVL C00525 V=800.0 PL=0
MOVL C00526 V=800.0 PL=0
MOVL C00527 V=800.0 PL=0
MOVL C00528 V=800.0 PL=0
MOVL C00529 V=800.0 PL=0
MOVL C00530 V=800.0 PL=0
MOVL C00531 V=800.0 PL=0
MOVL C00532 V=800.0 PL=0
MOVL C00533 V=800.0 PL=0
MOVL C00534 V=800.0 PL=0
MOVL C00535 V=800.0 PL=0
MOVL C00536 V=800.0 PL=0
MOVL C00537 V=800.0 PL=0
MOVL C00538 V=800.0 PL=0
MOVL C00539 V=800.0 PL=0
MOVL C00540 V=800.0 PL=0
MOVL C00541 V=800.0 PL=0
MOVL C00542 V=800.0 PL=0
MOVL C00543 V=800.0 PL=0
MOVL C00544 V=800.0 PL=0
MOVL C00545 V=800.0 PL=0
MOVL C00546 V=800.0 PL=0
MOVL C00547 V=800.0 PL=0
MOVL C00548 V=800.0 PL=0
MOVL C00549 V=800.0 PL=0
MOVL C00550 V=800.0 PL=0
MOVL C00551 V=800.0 PL=0
MOVL C00552 V=800.0 PL=0
MOVL C00553 V=800.0 PL=0
MOVL C00554 V=800.0 PL=0
MOVL C00555 V=800.0 PL=0
MOVL C00556 V=800.0 PL=0
MOVL C00557 V=800.0 PL=0
MOVL C00558 V=800.0 PL=0
MOVL C00559 V=800.0 PL=0
MOVL C00560 V=800.0 PL=0
MOVL C00561 V=800.0 PL=0
MOVL C00562 V=800.0 PL=0
MOVL C00563 V=800.0 PL=0
MOVL C00564 V=800.0 PL=0
MOVL C00565 V=800.0 PL=0
MOVL C00566 V=800.0 PL=0
MOVL C00567 V=800.0 PL=0
MOVL C00568 V=800.0 PL=0
MOVL C00569 V=800.0 PL=0
MOVL C00570 V=800.0 PL=0
MOVL C00571 V=800.0 PL=0
MOVL C00572 V=800.0 PL=0
MOVL C00573 V=800.0 PL=0
MOVL C00574 V=800.0 PL=0
MOVL C00575 V=800.0 PL=0
MOVL C00576 V=800.0 PL=0
MOVL C00577 V=800.0 PL=0
MOVL C00578 V=800.0 PL=0
MOVL C00579 V=800.0 PL=0
MOVL C00580 V=800.0 PL=0
MOVL C00581 V=800.0 PL=0
MOVL C00582 V=800.0 PL=0
MOVL C00583 V=800.0 PL=0
MOVL C00584 V=800.0 PL=0
MOVL C00585 V=800.0 PL=0
MOVL C00586 V=800.0 PL=0
MOVL C00587 V=800.0 PL=0
MOVL C00588 V=800.0 PL=0
MOVL C00589 V=800.0 PL=0
MOVL C00590 V=800.0 PL=0
MOVL C00591 V=800.0 PL=0
MOVL C00592 V=800.0 PL=0
MOVL C00593 V=800.0 PL=0
MOVL C00594 V=800.0 PL=0
MOVL C00595 V=800.0 PL=0
MOVL C00596 V=800.0 PL=0
MOVL C00597 V=800.0 PL=0
MOVL C00598 V=800.0 PL=0
MOVL C00599 V=800.0 PL=0
MOVL C00600 V=800.0 PL=0
MOVL C00601 V=800.0 PL=0
MOVL C00602 V=800.0 PL=0
MOVL C00603 V=800.0 PL=0
MOVL C00604 V=800.0 PL=0
MOVL C00605 V=800.0 PL=0
MOVL C00606 V=800.0 PL=0
MOVL C00607 V=800.0 PL=0
MOVL C00608 V=800.0 PL=0
MOVL C00609 V=800.0 PL=0
MOVL C00610 V=800.0 PL=0
MOVL C00611 V=800.0 PL=0
MOVL C00612 V=800.0 PL=0
MOVL C00613 V=800.0 PL=0
MOVL C00614 V=800.0 PL=0
MOVL C00615 V=800.0 PL=0
MOVL C00616 V=800.0 PL=0
MOVL C00617 V=800.0 PL=0
MOVL C00618 V=800.0 PL=0
MOVL C00619 V=800.0 PL=0
MOVL C00620 V=800.0 PL=0
MOVL C00621 V=800.0 PL=0
MOVL C00622 V=800.0 PL=0
MOVL C00623 V=800.0 PL=0
MOVL C00624 V=800.0 PL=0
MOVL C00625 V=800.0 PL=0
MOVL C00626 V=800.0 PL=0
MOVL C00627 V=800.0 PL=0
MOVL C00628 V=800.0 PL=0
MOVL C00629 V=800.0 PL=0
MOVL C00630 V=800.0 PL=0
MOVL C00631 V=800.0 PL=0
MOVL C00632 V=800.0 PL=0
MOVL C00633 V=800.0 PL=0
MOVL C00634 V=800.0 PL=0
MOVL C00635 V=800.0 PL=0
MOVL C00636 V=800.0 PL=0
MOVL C00637 V=800.0 PL=0
MOVL C00638 V=800.0 PL=0
MOVL C00639 V=800.0 PL=0
MOVL C00640 V=800.0 PL=0
MOVL C00641 V=800.0 PL=0
MOVL C00642 V=800.0 PL=0
MOVL C00643 V=800.0 PL=0
MOVL C00644 V=800.0 PL=0
MOVL C00645 V=800.0 PL=0
MOVL C00646 V=800.0 PL=0
MOVL C00647 V=800.0 PL=0
MOVL C00648 V=800.0 PL=0
MOVL C00649 V=800.0 PL=0
MOVL C00650 V=800.0 PL=0
MOVL C00651 V=800.0 PL=0
MOVL C00652 V=800.0 PL=0
MOVL C00653 V=800.0 PL=0
MOVL C00654 V=800.0 PL=0
MOVL C00655 V=800.0 PL=0
MOVL C00656 V=800.0 PL=0
MOVL C00657 V=800.0 PL=0
MOVL C00658 V=800.0 PL=0
MOVL C00659 V=800.0 PL=0
MOVL C00660 V=800.0 PL=0
MOVL C00661 V=800.0 PL=0
MOVL C00662 V=800.0 PL=0
MOVL C00663 V=800.0 PL=0
MOVL C00664 V=800.0 PL=0
MOVL C00665 V=800.0 PL=0
MOVL C00666 V=800.0 PL=0
MOVL C00667 V=800.0 PL=0
MOVL C00668 V=800.0 PL=0
MOVL C00669 V=800.0 PL=0
MOVL C00670 V=800.0 PL=0
MOVL C00671 V=800.0 PL=0
MOVL C00672 V=800.0 PL=0
MOVL C00673 V=800.0 PL=0
MOVL C00674 V=800.0 PL=0
MOVL C00675 V=800.0 PL=0
MOVL C00676 V=800.0 PL=0
MOVL C00677 V=800.0 PL=0
MOVL C00678 V=800.0 PL=0
MOVL C00679 V=800.0 PL=0
MOVL C00680 V=800.0 PL=0
MOVL C00681 V=800.0 PL=0
MOVL C00682 V=800.0 PL=0
MOVL C00683 V=800.0 PL=0
MOVL C00684 V=800.0 PL=0
MOVL C00685 V=800.0 PL=0
MOVL C00686 V=800.0 PL=0
MOVL C00687 V=800.0 PL=0
MOVL C00688 V=800.0 PL=0
MOVL C00689 V=800.0 PL=0
MOVL C00690 V=800.0 PL=0
MOVL C00691 V=800.0 PL=0
MOVL C00692 V=800.0 PL=0
MOVL C00693 V=800.0 PL=0
MOVL C00694 V=800.0 PL=0
MOVL C00695 V=800.0 PL=0
MOVL C00696 V=800.0 PL=0
MOVL C00697 V=800.0 PL=0
MOVL C00698 V=800.0 PL=0
MOVL C00699 V=800.0 PL=0
MOVL C00700 V=800.0 PL=0
MOVL C00701 V=800.0 PL=0
MOVL C00702 V=800.0 PL=0
MOVL C00703 V=800.0 PL=0
MOVL C00704 V=800.0 PL=0
MOVL C00705 V=800.0 PL=0
MOVL C00706 V=800.0 PL=0
MOVL C00707 V=800.0 PL=0
MOVL C00708 V=800.0 PL=0
MOVL C00709 V=800.0 PL=0
MOVL C00710 V=800.0 PL=0
MOVL C00711 V=800.0 PL=0
MOVL C00712 V=800.0 PL=0
MOVL C00713 V=800.0 PL=0
MOVL C00714 V=800.0 PL=0
MOVL C00715 V=800.0 PL=0
MOVL C00716 V=800.0 PL=0
MOVL C00717 V=800.0 PL=0
MOVL C00718 V=800.0 PL=0
MOVL C00719 V=800.0 PL=0
MOVL C00720 V=800.0 PL=0
MOVL C00721 V=800.0 PL=0
MOVL C00722 V=800.0 PL=0
MOVL C00723 V=800.0 PL=0
MOVL C00724 V=800.0 PL=0
MOVL C00725 V=800.0 PL=0
MOVL C00726 V=800.0 PL=0
MOVL C00727 V=800.0 PL=0
MOVL C00728 V=800.0 PL=0
MOVL C00729 V=800.0 PL=0
MOVL C00730 V=800.0 PL=0
MOVL C00731 V=800.0 PL=0
MOVL C00732 V=800.0 PL=0
MOVL C00733 V=800.0 PL=0
MOVL C00734 V=800.0 PL=0
MOVL C00735 V=800.0 PL=0
MOVL C00736 V=800.0 PL=0
MOVL C00737 V=800.0 PL=0
MOVL C00738 V=800.0 PL=0
MOVL C00739 V=800.0 PL=0
MOVL C00740 V=800.0 PL=0
MOVL C00741 V=800.0 PL=0
MOVL C00742 V=800.0 PL=0
MOVL C00743 V=800.0 PL=0
MOVL C00744 V=800.0 PL=0
MOVL C00745 V=800.0 PL=0
MOVL C00746 V=800.0 PL=0
MOVL C00747 V=800.0 PL=0
MOVL C00748 V=800.0 PL=0
MOVL C00749 V=800.0 PL=0
MOVL C00750 V=800.0 PL=0
MOVL C00751 V=800.0 PL=0
MOVL C00752 V=800.0 PL=0
MOVL C00753 V=800.0 PL=0
MOVL C00754 V=800.0 PL=0
MOVL C00755 V=800.0 PL=0
MOVL C00756 V=800.0 PL=0
MOVL C00757 V=800.0 PL=0
MOVL C00758 V=800.0 PL=0
MOVL C00759 V=800.0 PL=0
MOVL C00760 V=800.0 PL=0
MOVL C00761 V=800.0 PL=0
MOVL C00762 V=800.0 PL=0
MOVL C00763 V=800.0 PL=0
MOVL C00764 V=800.0 PL=0
MOVL C00765 V=800.0 PL=0
MOVL C00766 V=800.0 PL=0
MOVL C00767 V=800.0 PL=0
MOVL C00768 V=800.0 PL=0
MOVL C00769 V=800.0 PL=0
MOVL C00770 V=800.0 PL=0
MOVL C00771 V=800.0 PL=0
MOVL C00772 V=800.0 PL=0
MOVL C00773 V=800.0 PL=0
MOVL C00774 V=800.0 PL=0
MOVL C00775 V=800.0 PL=0
MOVL C00776 V=800.0 PL=0
MOVL C00777 V=800.0 PL=0
MOVL C00778 V=800.0 PL=0
MOVL C00779 V=800.0 PL=0
MOVL C00780 V=800.0 PL=0
MOVL C00781 V=800.0 PL=0
MOVL C00782 V=800.0 PL=0
MOVL C00783 V=800.0 PL=0
MOVL C00784 V=800.0 PL=0
MOVL C00785 V=800.0 PL=0
MOVL C00786 V=800.0 PL=0
MOVL C00787 V=800.0 PL=0
MOVL C00788 V=800.0 PL=0
MOVL C00789 V=800.0 PL=0
MOVL C00790 V=800.0 PL=0
MOVL C00791 V=800.0 PL=0
MOVL C00792 V=800.0 PL=0
MOVL C00793 V=800.0 PL=0
MOVL C00794 V=800.0 PL=0
MOVL C00795 V=800.0 PL=0
MOVL C00796 V=800.0 PL=0
MOVL C00797 V=800.0 PL=0
MOVL C00798 V=800.0 PL=0
MOVL C00799 V=800.0 PL=0
MOVL C00800 V=800.0 PL=0
MOVL C00801 V=800.0 PL=0
MOVL C00802 V=800.0 PL=0
MOVL C00803 V=800.0 PL=0
MOVL C00804 V=800.0 PL=0
MOVL C00805 V=800.0 PL=0
MOVL C00806 V=800.0 PL=0
MOVL C00807 V=800.0 PL=0
MOVL C00808 V=800.0 PL=0
MOVL C00809 V=800.0 PL=0
MOVL C00810 V=800.0 PL=0
MOVL C00811 V=800.0 PL=0
MOVL C00812 V=800.0 PL=0
MOVL C00813 V=800.0 PL=0
MOVL C00814 V=800.0 PL=0
MOVL C00815 V=800.0 PL=0
MOVL C00816 V=800.0 PL=0
MOVL C00817 V=800.0 PL=0
MOVL C00818 V=800.0 PL=0
MOVL C00819 V=800.0 PL=0
MOVL C00820 V=800.0 PL=0
MOVL C00821 V=800.0 PL=0
MOVL C00822 V=800.0 PL=0
MOVL C00823 V=800.0 PL=0
MOVL C00824 V=800.0 PL=0
MOVL C00825 V=800.0 PL=0
MOVL C00826 V=800.0 PL=0
MOVL C00827 V=800.0 PL=0
MOVL C00828 V=800.0 PL=0
MOVL C00829 V=800.0 PL=0
MOVL C00830 V=800.0 PL=0
MOVL C00831 V=800.0 PL=0
MOVL C00832 V=800.0 PL=0
MOVL C00833 V=800.0 PL=0
MOVL C00834 V=800.0 PL=0
MOVL C00835 V=800.0 PL=0
MOVL C00836 V=800.0 PL=0
MOVL C00837 V=800.0 PL=0
MOVL C00838 V=800.0 PL=0
MOVL C00839 V=800.0 PL=0
MOVL C00840 V=800.0 PL=0
MOVL C00841 V=800.0 PL=0
MOVL C00842 V=800.0 PL=0
MOVL C00843 V=800.0 PL=0
MOVL C00844 V=800.0 PL=0
MOVL C00845 V=800.0 PL=0
MOVL C00846 V=800.0 PL=0
MOVL C00847 V=800.0 PL=0
MOVL C00848 V=800.0 PL=0
MOVL C00849 V=800.0 PL=0
MOVL C00850 V=800.0 PL=0
MOVL C00851 V=800.0 PL=0
MOVL C00852 V=800.0 PL=0
MOVL C00853 V=800.0 PL=0
MOVL C00854 V=800.0 PL=0
MOVL C00855 V=800.0 PL=0
MOVL C00856 V=800.0 PL=0
MOVL C00857 V=800.0 PL=0
MOVL C00858 V=800.0 PL=0
MOVL C00859 V=800.0 PL=0
MOVL C00860 V=800.0 PL=0
MOVL C00861 V=800.0 PL=0
MOVL C00862 V=800.0 PL=0
MOVL C00863 V=800.0 PL=0
MOVL C00864 V=800.0 PL=0
MOVL C00865 V=800.0 PL=0
MOVL C00866 V=800.0 PL=0
MOVL C00867 V=800.0 PL=0
MOVL C00868 V=800.0 PL=0
MOVL C00869 V=800.0 PL=0
MOVL C00870 V=800.0 PL=0
MOVL C00871 V=800.0 PL=0
MOVL C00872 V=800.0 PL=0
MOVL C00873 V=800.0 PL=0
MOVL C00874 V=800.0 PL=0
MOVL C00875 V=800.0 PL=0
MOVL C00876 V=800.0 PL=0
MOVL C00877 V=800.0 PL=0
MOVL C00878 V=800.0 PL=0
MOVL C00879 V=800.0 PL=0
MOVL C00880 V=800.0 PL=0
MOVL C00881 V=800.0 PL=0
MOVL C00882 V=800.0 PL=0
MOVL C00883 V=800.0 PL=0
MOVL C00884 V=800.0 PL=0
MOVL C00885 V=800.0 PL=0
MOVL C00886 V=800.0 PL=0
MOVL C00887 V=800.0 PL=0
MOVL C00888 V=800.0 PL=0
MOVL C00889 V=800.0 PL=0
MOVL C00890 V=800.0 PL=0
MOVL C00891 V=800.0 PL=0
MOVL C00892 V=800.0 PL=0
MOVL C00893 V=800.0 PL=0
MOVL C00894 V=800.0 PL=0
MOVL C00895 V=800.0 PL=0
MOVL C00896 V=800.0 PL=0
MOVL C00897 V=800.0 PL=0
MOVL C00898 V=800.0 PL=0
MOVL C00899 V=800.0 PL=0
MOVL C00900 V=800.0 PL=0
MOVL C00901 V=800.0 PL=0
MOVL C00902 V=800.0 PL=0
MOVL C00903 V=800.0 PL=0
MOVL C00904 V=800.0 PL=0
MOVL C00905 V=800.0 PL=0
MOVL C00906 V=800.0 PL=0
MOVL C00907 V=800.0 PL=0
MOVL C00908 V=800.0 PL=0
MOVL C00909 V=800.0 PL=0
MOVL C00910 V=800.0 PL=0
MOVL C00911 V=800.0 PL=0
MOVL C00912 V=800.0 PL=0
MOVL C00913 V=800.0 PL=0
MOVL C00914 V=800.0 PL=0
MOVL C00915 V=800.0 PL=0
MOVL C00916 V=800.0 PL=0
MOVL C00917 V=800.0 PL=0
MOVL C00918 V=800.0 PL=0
MOVL C00919 V=800.0 PL=0
MOVL C00920 V=800.0 PL=0
MOVL C00921 V=800.0 PL=0
MOVL C00922 V=800.0 PL=0
MOVL C00923 V=800.0 PL=0
MOVL C00924 V=800.0 PL=0
MOVL C00925 V=800.0 PL=0
MOVL C00926 V=800.0 PL=0
MOVL C00927 V=800.0 PL=0
MOVL C00928 V=800.0 PL=0
MOVL C00929 V=800.0 PL=0
MOVL C00930 V=800.0 PL=0
MOVL C00931 V=800.0 PL=0
MOVL C00932 V=800.0 PL=0
MOVL C00933 V=800.0 PL=0
MOVL C00934 V=800.0 PL=0
MOVL C00935 V=800.0 PL=0
MOVL C00936 V=800.0 PL=0
MOVL C00937 V=800.0 PL=0
MOVL C00938 V=800.0 PL=0
MOVL C00939 V=800.0 PL=0
MOVL C00940 V=800.0 PL=0
MOVL C00941 V=800.0 PL=0
MOVL C00942 V=800.0 PL=0
MOVL C00943 V=800.0 PL=0
MOVL C00944 V=800.0 PL=0
MOVL C00945 V=800.0 PL=0
MOVL C00946 V=800.0 PL=0
MOVL C00947 V=800.0 PL=0
MOVL C00948 V=800.0 PL=0
MOVL C00949 V=800.0 PL=0
MOVL C00950 V=800.0 PL=0
MOVL C00951 V=800.0 PL=0
MOVL C00952 V=800.0 PL=0
MOVL C00953 V=800.0 PL=0
MOVL C00954 V=800.0 PL=0
MOVL C00955 V=800.0 PL=0
MOVL C00956 V=800.0 PL=0
MOVL C00957 V=800.0 PL=0
MOVL C00958 V=800.0 PL=0
MOVL C00959 V=800.0 PL=0
MOVL C00960 V=800.0 PL=0
MOVL C00961 V=800.0 PL=0
MOVL C00962 V=800.0 PL=0
MOVL C00963 V=800.0 PL=0
MOVL C00964 V=800.0 PL=0
MOVL C00965 V=800.0 PL=0
MOVL C00966 V=800.0 PL=0
MOVL C00967 V=800.0 PL=0
MOVL C00968 V=800.0 PL=0
MOVL C00969 V=800.0 PL=0
MOVL C00970 V=800.0 PL=0
MOVL C00971 V=800.0 PL=0
MOVL C00972 V=800.0 PL=0
MOVL C00973 V=800.0 PL=0
MOVL C00974 V=800.0 PL=0
MOVL C00975 V=800.0 PL=0
MOVL C00976 V=800.0 PL=0
MOVL C00977 V=800.0 PL=0
MOVL C00978 V=800.0 PL=0
MOVL C00979 V=800.0 PL=0
MOVL C00980 V=800.0 PL=0
MOVL C00981 V=800.0 PL=0
MOVL C00982 V=800.0 PL=0
MOVL C00983 V=800.0 PL=0
MOVL C00984 V=800.0 PL=0
MOVL C00985 V=800.0 PL=0
MOVL C00986 V=800.0 PL=0
MOVL C00987 V=800.0 PL=0
MOVL C00988 V=800.0 PL=0
MOVL C00989 V=800.0 PL=0
MOVL C00990 V=800.0 PL=0
MOVL C00991 V=800.0 PL=0
MOVL C00992 V=800.0 PL=0
MOVL C00993 V=800.0 PL=0
MOVL C00994 V=800.0 PL=0
MOVL C00995 V=800.0 PL=0
MOVL C00996 V=800.0 PL=0
MOVL C00997 V=800.0 PL=0
MOVL C00998 V=800.0 PL=0
MOVL C00999 V=800.0 PL=0
MOVL C01000 V=800.0 PL=0
MOVL C01001 V=800.0 PL=0
MOVL C01002 V=800.0 PL=0
MOVL C01003 V=800.0 PL=0
MOVL C01004 V=800.0 PL=0
MOVL C01005 V=800.0 PL=0
MOVL C01006 V=800.0 PL=0
MOVL C01007 V=800.0 PL=0
MOVL C01008 V=800.0 PL=0
MOVL C01009 V=800.0 PL=0
MOVL C01010 V=800.0 PL=0
MOVL C01011 V=800.0 PL=0
MOVL C01012 V=800.0 PL=0
MOVL C01013 V=800.0 PL=0
MOVL C01014 V=800.0 PL=0
MOVL C01015 V=800.0 PL=0
MOVL C01016 V=800.0 PL=0
MOVL C01017 V=800.0 PL=0
MOVL C01018 V=800.0 PL=0
MOVL C01019 V=800.0 PL=0
MOVL C01020 V=800.0 PL=0
MOVL C01021 V=800.0 PL=0
MOVL C01022 V=800.0 PL=0
MOVL C01023 V=800.0 PL=0
MOVL C01024 V=800.0 PL=0
MOVL C01025 V=800.0 PL=0
MOVL C01026 V=800.0 PL=0
MOVL C01027 V=800.0 PL=0
MOVL C01028 V=800.0 PL=0
MOVL C01029 V=800.0 PL=0
MOVL C01030 V=800.0 PL=0
MOVL C01031 V=800.0 PL=0
MOVL C01032 V=800.0 PL=0
MOVL C01033 V=800.0 PL=0
MOVL C01034 V=800.0 PL=0
MOVL C01035 V=800.0 PL=0
MOVL C01036 V=800.0 PL=0
MOVL C01037 V=800.0 PL=0
MOVL C01038 V=800.0 PL=0
MOVL C01039 V=800.0 PL=0
MOVL C01040 V=800.0 PL=0
MOVL C01041 V=800.0 PL=0
MOVL C01042 V=800.0 PL=0
MOVL C01043 V=800.0 PL=0
MOVL C01044 V=800.0 PL=0
MOVL C01045 V=800.0 PL=0
MOVL C01046 V=800.0 PL=0
MOVL C01047 V=800.0 PL=0
MOVL C01048 V=800.0 PL=0
MOVL C01049 V=800.0 PL=0
MOVL C01050 V=800.0 PL=0
MOVL C01051 V=800.0 PL=0
MOVL C01052 V=800.0 PL=0
MOVL C01053 V=800.0 PL=0
MOVL C01054 V=800.0 PL=0
MOVL C01055 V=800.0 PL=0
MOVL C01056 V=800.0 PL=0
MOVL C01057 V=800.0 PL=0
MOVL C01058 V=800.0 PL=0
MOVL C01059 V=800.0 PL=0
MOVL C01060 V=800.0 PL=0
MOVL C01061 V=800.0 PL=0
MOVL C01062 V=800.0 PL=0
MOVL C01063 V=800.0 PL=0
MOVL C01064 V=800.0 PL=0
MOVL C01065 V=800.0 PL=0
MOVL C01066 V=800.0 PL=0
MOVL C01067 V=800.0 PL=0
MOVL C01068 V=800.0 PL=0
MOVL C01069 V=800.0 PL=0
MOVL C01070 V=800.0 PL=0
MOVL C01071 V=800.0 PL=0
MOVL C01072 V=800.0 PL=0
MOVL C01073 V=800.0 PL=0
MOVL C01074 V=800.0 PL=0
MOVL C01075 V=800.0 PL=0
MOVL C01076 V=800.0 PL=0
MOVL C01077 V=800.0 PL=0
MOVL C01078 V=800.0 PL=0
MOVL C01079 V=800.0 PL=0
MOVL C01080 V=800.0 PL=0
MOVL C01081 V=800.0 PL=0
MOVL C01082 V=800.0 PL=0
MOVL C01083 V=800.0 PL=0
MOVL C01084 V=800.0 PL=0
MOVL C01085 V=800.0 PL=0
MOVL C01086 V=800.0 PL=0
MOVL C01087 V=800.0 PL=0
MOVL C01088 V=800.0 PL=0
MOVL C01089 V=800.0 PL=0
MOVL C01090 V=800.0 PL=0
MOVL C01091 V=800.0 PL=0
MOVL C01092 V=800.0 PL=0
MOVL C01093 V=800.0 PL=0
MOVL C01094 V=800.0 PL=0
MOVL C01095 V=800.0 PL=0
MOVL C01096 V=800.0 PL=0
MOVL C01097 V=800.0 PL=0
MOVL C01098 V=800.0 PL=0
MOVL C01099 V=800.0 PL=0
MOVL C01100 V=800.0 PL=0
MOVL C01101 V=800.0 PL=0
MOVL C01102 V=800.0 PL=0
MOVL C01103 V=800.0 PL=0
MOVL C01104 V=800.0 PL=0
MOVL C01105 V=800.0 PL=0
MOVL C01106 V=800.0 PL=0
MOVL C01107 V=800.0 PL=0
MOVL C01108 V=800.0 PL=0
MOVL C01109 V=800.0 PL=0
MOVL C01110 V=800.0 PL=0
MOVL C01111 V=800.0 PL=0
MOVL C01112 V=800.0 PL=0
MOVL C01113 V=800.0 PL=0
MOVL C01114 V=800.0 PL=0
MOVL C01115 V=800.0 PL=0
MOVL C01116 V=800.0 PL=0
MOVL C01117 V=800.0 PL=0
MOVL C01118 V=800.0 PL=0
MOVL C01119 V=800.0 PL=0
MOVL C01120 V=800.0 PL=0
MOVL C01121 V=800.0 PL=0
MOVL C01122 V=800.0 PL=0
MOVL C01123 V=800.0 PL=0
MOVL C01124 V=800.0 PL=0
MOVL C01125 V=800.0 PL=0
MOVL C01126 V=800.0 PL=0
MOVL C01127 V=800.0 PL=0
MOVL C01128 V=800.0 PL=0
MOVL C01129 V=800.0 PL=0
MOVL C01130 V=800.0 PL=0
MOVL C01131 V=800.0 PL=0
MOVL C01132 V=800.0 PL=0
MOVL C01133 V=800.0 PL=0
MOVL C01134 V=800.0 PL=0
MOVL C01135 V=800.0 PL=0
MOVL C01136 V=800.0 PL=0
MOVL C01137 V=800.0 PL=0
MOVL C01138 V=800.0 PL=0
MOVL C01139 V=800.0 PL=0
MOVL C01140 V=800.0 PL=0
MOVL C01141 V=800.0 PL=0
MOVL C01142 V=800.0 PL=0
MOVL C01143 V=800.0 PL=0
MOVL C01144 V=800.0 PL=0
MOVL C01145 V=800.0 PL=0
MOVL C01146 V=800.0 PL=0
MOVL C01147 V=800.0 PL=0
MOVL C01148 V=800.0 PL=0
MOVL C01149 V=800.0 PL=0
MOVL C01150 V=800.0 PL=0
MOVL C01151 V=800.0 PL=0
MOVL C01152 V=800.0 PL=0
MOVL C01153 V=800.0 PL=0
MOVL C01154 V=800.0 PL=0
MOVL C01155 V=800.0 PL=0
MOVL C01156 V=800.0 PL=0
MOVL C01157 V=800.0 PL=0
MOVL C01158 V=800.0 PL=0
MOVL C01159 V=800.0 PL=0
MOVL C01160 V=800.0 PL=0
MOVL C01161 V=800.0 PL=0
MOVL C01162 V=800.0 PL=0
MOVL C01163 V=800.0 PL=0
MOVL C01164 V=800.0 PL=0
MOVL C01165 V=800.0 PL=0
MOVL C01166 V=800.0 PL=0
MOVL C01167 V=800.0 PL=0
MOVL C01168 V=800.0 PL=0
MOVL C01169 V=800.0 PL=0
MOVL C01170 V=800.0 PL=0
MOVL C01171 V=800.0 PL=0
MOVL C01172 V=800.0 PL=0
MOVL C01173 V=800.0 PL=0
MOVL C01174 V=800.0 PL=0
MOVL C01175 V=800.0 PL=0
MOVL C01176 V=800.0 PL=0
MOVL C01177 V=800.0 PL=0
MOVL C01178 V=800.0 PL=0
MOVL C01179 V=800.0 PL=0
MOVL C01180 V=800.0 PL=0
MOVL C01181 V=800.0 PL=0
MOVL C01182 V=800.0 PL=0
MOVL C01183 V=800.0 PL=0
MOVL C01184 V=800.0 PL=0
MOVL C01185 V=800.0 PL=0
MOVL C01186 V=800.0 PL=0
MOVL C01187 V=800.0 PL=0
MOVL C01188 V=800.0 PL=0
MOVL C01189 V=800.0 PL=0
MOVL C01190 V=800.0 PL=0
MOVL C01191 V=800.0 PL=0
MOVL C01192 V=800.0 PL=0
MOVL C01193 V=800.0 PL=0
MOVL C01194 V=800.0 PL=0
MOVL C01195 V=800.0 PL=0
MOVL C01196 V=800.0 PL=0
MOVL C01197 V=800.0 PL=0
MOVL C01198 V=800.0 PL=0
MOVL C01199 V=800.0 PL=0
MOVL C01200 V=800.0 PL=0
MOVL C01201 V=800.0 PL=0
MOVL C01202 V=800.0 PL=0
MOVL C01203 V=800.0 PL=0
MOVL C01204 V=800.0 PL=0
MOVL C01205 V=800.0 PL=0
MOVL C01206 V=800.0 PL=0
MOVL C01207 V=800.0 PL=0
MOVL C01208 V=800.0 PL=0
MOVL C01209 V=800.0 PL=0
MOVL C01210 V=800.0 PL=0
MOVL C01211 V=800.0 PL=0
MOVL C01212 V=800.0 PL=0
MOVL C01213 V=800.0 PL=0
MOVL C01214 V=800.0 PL=0
MOVL C01215 V=800.0 PL=0
MOVL C01216 V=800.0 PL=0
MOVL C01217 V=800.0 PL=0
MOVL C01218 V=800.0 PL=0
MOVL C01219 V=800.0 PL=0
MOVL C01220 V=800.0 PL=0
MOVL C01221 V=800.0 PL=0
MOVL C01222 V=800.0 PL=0
MOVL C01223 V=800.0 PL=0
MOVL C01224 V=800.0 PL=0
MOVL C01225 V=800.0 PL=0
MOVL C01226 V=800.0 PL=0
MOVL C01227 V=800.0 PL=0
MOVL C01228 V=800.0 PL=0
MOVL C01229 V=800.0 PL=0
MOVL C01230 V=800.0 PL=0
MOVL C01231 V=800.0 PL=0
MOVL C01232 V=800.0 PL=0
MOVL C01233 V=800.0 PL=0
MOVL C01234 V=800.0 PL=0
MOVL C01235 V=800.0 PL=0
MOVL C01236 V=800.0 PL=0
MOVL C01237 V=800.0 PL=0
MOVL C01238 V=800.0 PL=0
MOVL C01239 V=800.0 PL=0
MOVL C01240 V=800.0 PL=0
MOVL C01241 V=800.0 PL=0
MOVL C01242 V=800.0 PL=0
MOVL C01243 V=800.0 PL=0
MOVL C01244 V=800.0 PL=0
MOVL C01245 V=800.0 PL=0
MOVL C01246 V=800.0 PL=0
MOVL C01247 V=800.0 PL=0
MOVL C01248 V=800.0 PL=0
MOVL C01249 V=800.0 PL=0
MOVL C01250 V=800.0 PL=0
MOVL C01251 V=800.0 PL=0
MOVL C01252 V=800.0 PL=0
MOVL C01253 V=800.0 PL=0
MOVL C01254 V=800.0 PL=0
MOVL C01255 V=800.0 PL=0
MOVL C01256 V=800.0 PL=0
MOVL C01257 V=800.0 PL=0
MOVL C01258 V=800.0 PL=0
MOVL C01259 V=800.0 PL=0
MOVL C01260 V=800.0 PL=0
MOVL C01261 V=800.0 PL=0
MOVL C01262 V=800.0 PL=0
MOVL C01263 V=800.0 PL=0
MOVL C01264 V=800.0 PL=0
MOVL C01265 V=800.0 PL=0
MOVL C01266 V=800.0 PL=0
MOVL C01267 V=800.0 PL=0
MOVL C01268 V=800.0 PL=0
MOVL C01269 V=800.0 PL=0
MOVL C01270 V=800.0 PL=0
MOVL C01271 V=800.0 PL=0
MOVL C01272 V=800.0 PL=0
MOVL C01273 V=800.0 PL=0
MOVL C01274 V=800.0 PL=0
MOVL C01275 V=800.0 PL=0
MOVL C01276 V=800.0 PL=0
MOVL C01277 V=800.0 PL=0
MOVL C01278 V=800.0 PL=0
MOVL C01279 V=800.0 PL=0
MOVL C01280 V=800.0 PL=0
MOVL C01281 V=800.0 PL=0
MOVL C01282 V=800.0 PL=0
MOVL C01283 V=800.0 PL=0
MOVL C01284 V=800.0 PL=0
MOVL C01285 V=800.0 PL=0
MOVL C01286 V=800.0 PL=0
MOVL C01287 V=800.0 PL=0
MOVL C01288 V=800.0 PL=0
MOVL C01289 V=800.0 PL=0
MOVL C01290 V=800.0 PL=0
MOVL C01291 V=800.0 PL=0
MOVL C01292 V=800.0 PL=0
MOVL C01293 V=800.0 PL=0
MOVL C01294 V=800.0 PL=0
MOVL C01295 V=800.0 PL=0
MOVL C01296 V=800.0 PL=0
MOVL C01297 V=800.0 PL=0
MOVL C01298 V=800.0 PL=0
MOVL C01299 V=800.0 PL=0
MOVL C01300 V=800.0 PL=0
MOVL C01301 V=800.0 PL=0
MOVL C01302 V=800.0 PL=0
MOVL C01303 V=800.0 PL=0
MOVL C01304 V=800.0 PL=0
MOVL C01305 V=800.0 PL=0
MOVL C01306 V=800.0 PL=0
MOVL C01307 V=800.0 PL=0
MOVL C01308 V=800.0 PL=0
MOVL C01309 V=800.0 PL=0
MOVL C01310 V=800.0 PL=0
MOVL C01311 V=800.0 PL=0
MOVL C01312 V=800.0 PL=0
MOVL C01313 V=800.0 PL=0
MOVL C01314 V=800.0 PL=0
MOVL C01315 V=800.0 PL=0
MOVL C01316 V=800.0 PL=0
MOVL C01317 V=800.0 PL=0
MOVL C01318 V=800.0 PL=0
MOVL C01319 V=800.0 PL=0
MOVL C01320 V=800.0 PL=0
MOVL C01321 V=800.0 PL=0
MOVL C01322 V=800.0 PL=0
MOVL C01323 V=800.0 PL=0
MOVL C01324 V=800.0 PL=0
MOVL C01325 V=800.0 PL=0
MOVL C01326 V=800.0 PL=0
MOVL C01327 V=800.0 PL=0
MOVL C01328 V=800.0 PL=0
MOVL C01329 V=800.0 PL=0
MOVL C01330 V=800.0 PL=0
MOVL C01331 V=800.0 PL=0
MOVL C01332 V=800.0 PL=0
MOVL C01333 V=800.0 PL=0
MOVL C01334 V=800.0 PL=0
MOVL C01335 V=800.0 PL=0
MOVL C01336 V=800.0 PL=0
MOVL C01337 V=800.0 PL=0
MOVL C01338 V=800.0 PL=0
MOVL C01339 V=800.0 PL=0
MOVL C01340 V=800.0 PL=0
MOVL C01341 V=800.0 PL=0
MOVL C01342 V=800.0 PL=0
MOVL C01343 V=800.0 PL=0
MOVL C01344 V=800.0 PL=0
MOVL C01345 V=800.0 PL=0
MOVL C01346 V=800.0 PL=0
MOVL C01347 V=800.0 PL=0
MOVL C01348 V=800.0 PL=0
MOVL C01349 V=800.0 PL=0
MOVL C01350 V=800.0 PL=0
MOVL C01351 V=800.0 PL=0
MOVL C01352 V=800.0 PL=0
MOVL C01353 V=800.0 PL=0
MOVL C01354 V=800.0 PL=0
MOVL C01355 V=800.0 PL=0
MOVL C01356 V=800.0 PL=0
MOVL C01357 V=800.0 PL=0
MOVL C01358 V=800.0 PL=0
MOVL C01359 V=800.0 PL=0
MOVL C01360 V=800.0 PL=0
MOVL C01361 V=800.0 PL=0
MOVL C01362 V=800.0 PL=0
MOVL C01363 V=800.0 PL=0
MOVL C01364 V=800.0 PL=0
MOVL C01365 V=800.0 PL=0
MOVL C01366 V=800.0 PL=0
MOVL C01367 V=800.0 PL=0
MOVL C01368 V=800.0 PL=0
MOVL C01369 V=800.0 PL=0
MOVL C01370 V=800.0 PL=0
MOVL C01371 V=800.0 PL=0
MOVL C01372 V=800.0 PL=0
MOVL C01373 V=800.0 PL=0
MOVL C01374 V=800.0 PL=0
MOVL C01375 V=800.0 PL=0
MOVL C01376 V=800.0 PL=0
MOVL C01377 V=800.0 PL=0
MOVL C01378 V=800.0 PL=0
MOVL C01379 V=800.0 PL=0
MOVL C01380 V=800.0 PL=0
MOVL C01381 V=800.0 PL=0
MOVL C01382 V=800.0 PL=0
MOVL C01383 V=800.0 PL=0
MOVL C01384 V=800.0 PL=0
MOVL C01385 V=800.0 PL=0
MOVL C01386 V=800.0 PL=0
MOVL C01387 V=800.0 PL=0
MOVL C01388 V=800.0 PL=0
MOVL C01389 V=800.0 PL=0
MOVL C01390 V=800.0 PL=0
MOVL C01391 V=800.0 PL=0
MOVL C01392 V=800.0 PL=0
MOVL C01393 V=800.0 PL=0
MOVL C01394 V=800.0 PL=0
MOVL C01395 V=800.0 PL=0
MOVL C01396 V=800.0 PL=0
MOVL C01397 V=800.0 PL=0
MOVL C01398 V=800.0 PL=0
MOVL C01399 V=800.0 PL=0
MOVL C01400 V=800.0 PL=0
MOVL C01401 V=800.0 PL=0
MOVL C01402 V=800.0 PL=0
MOVL C01403 V=800.0 PL=0
MOVL C01404 V=800.0 PL=0
MOVL C01405 V=800.0 PL=0
MOVL C01406 V=800.0 PL=0
MOVL C01407 V=800.0 PL=0
MOVL C01408 V=800.0 PL=0
MOVL C01409 V=800.0 PL=0
MOVL C01410 V=800.0 PL=0
MOVL C01411 V=800.0 PL=0
MOVL C01412 V=800.0 PL=0
MOVL C01413 V=800.0 PL=0
MOVL C01414 V=800.0 PL=0
MOVL C01415 V=800.0 PL=0
MOVL C01416 V=800.0 PL=0
MOVL C01417 V=800.0 PL=0
MOVL C01418 V=800.0 PL=0
MOVL C01419 V=800.0 PL=0
MOVL C01420 V=800.0 PL=0
MOVL C01421 V=800.0 PL=0
MOVL C01422 V=800.0 PL=0
MOVL C01423 V=800.0 PL=0
MOVL C01424 V=800.0 PL=0
MOVL C01425 V=800.0 PL=0
MOVL C01426 V=800.0 PL=0
MOVL C01427 V=800.0 PL=0
MOVL C01428 V=800.0 PL=0
MOVL C01429 V=800.0 PL=0
MOVL C01430 V=800.0 PL=0
MOVL C01431 V=800.0 PL=0
MOVL C01432 V=800.0 PL=0
MOVL C01433 V=800.0 PL=0
MOVL C01434 V=800.0 PL=0
MOVL C01435 V=800.0 PL=0
MOVL C01436 V=800.0 PL=0
MOVL C01437 V=800.0 PL=0
MOVL C01438 V=800.0 PL=0
MOVL C01439 V=800.0 PL=0
MOVL C01440 V=800.0 PL=0
MOVL C01441 V=800.0 PL=0
MOVL C01442 V=800.0 PL=0
MOVL C01443 V=800.0 PL=0
MOVL C01444 V=800.0 PL=0
MOVL C01445 V=800.0 PL=0
MOVL C01446 V=800.0 PL=0
MOVL C01447 V=800.0 PL=0
MOVL C01448 V=800.0 PL=0
MOVL C01449 V=800.0 PL=0
MOVL C01450 V=800.0 PL=0
MOVL C01451 V=800.0 PL=0
MOVL C01452 V=800.0 PL=0
MOVL C01453 V=800.0 PL=0
MOVL C01454 V=800.0 PL=0
MOVL C01455 V=800.0 PL=0
MOVL C01456 V=800.0 PL=0
MOVL C01457 V=800.0 PL=0
MOVL C01458 V=800.0 PL=0
MOVL C01459 V=800.0 PL=0
MOVL C01460 V=800.0 PL=0
MOVL C01461 V=800.0 PL=0
MOVL C01462 V=800.0 PL=0
MOVL C01463 V=800.0 PL=0
MOVL C01464 V=800.0 PL=0
MOVL C01465 V=800.0 PL=0
MOVL C01466 V=800.0 PL=0
MOVL C01467 V=800.0 PL=0
MOVL C01468 V=800.0 PL=0
MOVL C01469 V=800.0 PL=0
MOVL C01470 V=800.0 PL=0
MOVL C01471 V=800.0 PL=0
MOVL C01472 V=800.0 PL=0
MOVL C01473 V=800.0 PL=0
MOVL C01474 V=800.0 PL=0
MOVL C01475 V=800.0 PL=0
MOVL C01476 V=800.0 PL=0
MOVL C01477 V=800.0 PL=0
MOVL C01478 V=800.0 PL=0
MOVL C01479 V=800.0 PL=0
MOVL C01480 V=800.0 PL=0
MOVL C01481 V=800.0 PL=0
MOVL C01482 V=800.0 PL=0
MOVL C01483 V=800.0 PL=0
MOVL C01484 V=800.0 PL=0
MOVL C01485 V=800.0 PL=0
MOVL C01486 V=800.0 PL=0
MOVL C01487 V=800.0 PL=0
MOVL C01488 V=800.0 PL=0
MOVL C01489 V=800.0 PL=0
MOVL C01490 V=800.0 PL=0
MOVL C01491 V=800.0 PL=0
MOVL C01492 V=800.0 PL=0
MOVL C01493 V=800.0 PL=0
MOVL C01494 V=800.0 PL=0
MOVL C01495 V=800.0 PL=0
MOVL C01496 V=800.0 PL=0
MOVL C01497 V=800.0 PL=0
MOVL C01498 V=800.0 PL=0
MOVL C01499 V=800.0 PL=0
MOVL C01500 V=800.0 PL=0
MOVL C01501 V=800.0 PL=0
MOVL C01502 V=800.0 PL=0
MOVL C01503 V=800.0 PL=0
MOVL C01504 V=800.0 PL=0
MOVL C01505 V=800.0 PL=0
MOVL C01506 V=800.0 PL=0
MOVL C01507 V=800.0 PL=0
MOVL C01508 V=800.0 PL=0
MOVL C01509 V=800.0 PL=0
MOVL C01510 V=800.0 PL=0
MOVL C01511 V=800.0 PL=0
MOVL C01512 V=800.0 PL=0
MOVL C01513 V=800.0 PL=0
MOVL C01514 V=800.0 PL=0
MOVL C01515 V=800.0 PL=0
MOVL C01516 V=800.0 PL=0
MOVL C01517 V=800.0 PL=0
MOVL C01518 V=800.0 PL=0
MOVL C01519 V=800.0 PL=0
MOVL C01520 V=800.0 PL=0
MOVL C01521 V=800.0 PL=0
MOVL C01522 V=800.0 PL=0
MOVL C01523 V=800.0 PL=0
MOVL C01524 V=800.0 PL=0
MOVL C01525 V=800.0 PL=0
MOVL C01526 V=800.0 PL=0
MOVL C01527 V=800.0 PL=0
MOVL C01528 V=800.0 PL=0
MOVL C01529 V=800.0 PL=0
MOVL C01530 V=800.0 PL=0
MOVL C01531 V=800.0 PL=0
MOVL C01532 V=800.0 PL=0
MOVL C01533 V=800.0 PL=0
MOVL C01534 V=800.0 PL=0
MOVL C01535 V=800.0 PL=0
MOVL C01536 V=800.0 PL=0
MOVL C01537 V=800.0 PL=0
MOVL C01538 V=800.0 PL=0
MOVL C01539 V=800.0 PL=0
MOVL C01540 V=800.0 PL=0
MOVL C01541 V=800.0 PL=0
MOVL C01542 V=800.0 PL=0
MOVL C01543 V=800.0 PL=0
MOVL C01544 V=800.0 PL=0
MOVL C01545 V=800.0 PL=0
MOVL C01546 V=800.0 PL=0
MOVL C01547 V=800.0 PL=0
MOVL C01548 V=800.0 PL=0
MOVL C01549 V=800.0 PL=0
MOVL C01550 V=800.0 PL=0
MOVL C01551 V=800.0 PL=0
MOVL C01552 V=800.0 PL=0
MOVL C01553 V=800.0 PL=0
MOVL C01554 V=800.0 PL=0
MOVL C01555 V=800.0 PL=0
MOVL C01556 V=800.0 PL=0
MOVL C01557 V=800.0 PL=0
MOVL C01558 V=800.0 PL=0
MOVL C01559 V=800.0 PL=0
MOVL C01560 V=800.0 PL=0
MOVL C01561 V=800.0 PL=0
MOVL C01562 V=800.0 PL=0
MOVL C01563 V=800.0 PL=0
MOVL C01564 V=800.0 PL=0
MOVL C01565 V=800.0 PL=0
MOVL C01566 V=800.0 PL=0
MOVL C01567 V=800.0 PL=0
MOVL C01568 V=800.0 PL=0
MOVL C01569 V=800.0 PL=0
MOVL C01570 V=800.0 PL=0
MOVL C01571 V=800.0 PL=0
MOVL C01572 V=800.0 PL=0
MOVL C01573 V=800.0 PL=0
MOVL C01574 V=800.0 PL=0
MOVL C01575 V=800.0 PL=0
MOVL C01576 V=800.0 PL=0
MOVL C01577 V=800.0 PL=0
MOVL C01578 V=800.0 PL=0
MOVL C01579 V=800.0 PL=0
MOVL C01580 V=800.0 PL=0
MOVL C01581 V=800.0 PL=0
MOVL C01582 V=800.0 PL=0
MOVL C01583 V=800.0 PL=0
MOVL C01584 V=800.0 PL=0
MOVL C01585 V=800.0 PL=0
MOVL C01586 V=800.0 PL=0
MOVL C01587 V=800.0 PL=0
MOVL C01588 V=800.0 PL=0
MOVL C01589 V=800.0 PL=0
MOVL C01590 V=800.0 PL=0
MOVL C01591 V=800.0 PL=0
MOVL C01592 V=800.0 PL=0
MOVL C01593 V=800.0 PL=0
MOVL C01594 V=800.0 PL=0
MOVL C01595 V=800.0 PL=0
MOVL C01596 V=800.0 PL=0
MOVL C01597 V=800.0 PL=0
MOVL C01598 V=800.0 PL=0
MOVL C01599 V=800.0 PL=0
MOVL C01600 V=800.0 PL=0
MOVL C01601 V=800.0 PL=0
MOVL C01602 V=800.0 PL=0
MOVL C01603 V=800.0 PL=0
MOVL C01604 V=800.0 PL=0
MOVL C01605 V=800.0 PL=0
MOVL C01606 V=800.0 PL=0
MOVL C01607 V=800.0 PL=0
MOVL C01608 V=800.0 PL=0
MOVL C01609 V=800.0 PL=0
MOVL C01610 V=800.0 PL=0
MOVL C01611 V=800.0 PL=0
MOVL C01612 V=800.0 PL=0
MOVL C01613 V=800.0 PL=0
MOVL C01614 V=800.0 PL=0
MOVL C01615 V=800.0 PL=0
MOVL C01616 V=800.0 PL=0
MOVL C01617 V=800.0 PL=0
MOVL C01618 V=800.0 PL=0
MOVL C01619 V=800.0 PL=0
MOVL C01620 V=800.0 PL=0
MOVL C01621 V=800.0 PL=0
MOVL C01622 V=800.0 PL=0
MOVL C01623 V=800.0 PL=0
MOVL C01624 V=800.0 PL=0
MOVL C01625 V=800.0 PL=0
MOVL C01626 V=800.0 PL=0
MOVL C01627 V=800.0 PL=0
MOVL C01628 V=800.0 PL=0
MOVL C01629 V=800.0 PL=0
MOVL C01630 V=800.0 PL=0
MOVL C01631 V=800.0 PL=0
MOVL C01632 V=800.0 PL=0
MOVL C01633 V=800.0 PL=0
MOVL C01634 V=800.0 PL=0
MOVL C01635 V=800.0 PL=0
MOVL C01636 V=800.0 PL=0
MOVL C01637 V=800.0 PL=0
MOVL C01638 V=800.0 PL=0
MOVL C01639 V=800.0 PL=0
MOVL C01640 V=800.0 PL=0
MOVL C01641 V=800.0 PL=0
MOVL C01642 V=800.0 PL=0
MOVL C01643 V=800.0 PL=0
MOVL C01644 V=800.0 PL=0
MOVL C01645 V=800.0 PL=0
MOVL C01646 V=800.0 PL=0
MOVL C01647 V=800.0 PL=0
MOVL C01648 V=800.0 PL=0
MOVL C01649 V=800.0 PL=0
MOVL C01650 V=800.0 PL=0
MOVL C01651 V=800.0 PL=0
MOVL C01652 V=800.0 PL=0
MOVL C01653 V=800.0 PL=0
MOVL C01654 V=800.0 PL=0
MOVL C01655 V=800.0 PL=0
MOVL C01656 V=800.0 PL=0
MOVL C01657 V=800.0 PL=0
MOVL C01658 V=800.0 PL=0
MOVL C01659 V=800.0 PL=0
MOVL C01660 V=800.0 PL=0
MOVL C01661 V=800.0 PL=0
MOVL C01662 V=800.0 PL=0
MOVL C01663 V=800.0 PL=0
MOVL C01664 V=800.0 PL=0
MOVL C01665 V=800.0 PL=0
MOVL C01666 V=800.0 PL=0
MOVL C01667 V=800.0 PL=0
MOVL C01668 V=800.0 PL=0
MOVL C01669 V=800.0 PL=0
MOVL C01670 V=800.0 PL=0
MOVL C01671 V=800.0 PL=0
MOVL C01672 V=800.0 PL=0
MOVL C01673 V=800.0 PL=0
MOVL C01674 V=800.0 PL=0
MOVL C01675 V=800.0 PL=0
MOVL C01676 V=800.0 PL=0
MOVL C01677 V=800.0 PL=0
MOVL C01678 V=800.0 PL=0
MOVL C01679 V=800.0 PL=0
MOVL C01680 V=800.0 PL=0
MOVL C01681 V=800.0 PL=0
MOVL C01682 V=800.0 PL=0
MOVL C01683 V=800.0 PL=0
MOVL C01684 V=800.0 PL=0
MOVL C01685 V=800.0 PL=0
MOVL C01686 V=800.0 PL=0
MOVL C01687 V=800.0 PL=0
MOVL C01688 V=800.0 PL=0
MOVL C01689 V=800.0 PL=0
MOVL C01690 V=800.0 PL=0
MOVL C01691 V=800.0 PL=0
MOVL C01692 V=800.0 PL=0
MOVL C01693 V=800.0 PL=0
MOVL C01694 V=800.0 PL=0
MOVL C01695 V=800.0 PL=0
MOVL C01696 V=800.0 PL=0
MOVL C01697 V=800.0 PL=0
MOVL C01698 V=800.0 PL=0
MOVL C01699 V=800.0 PL=0
MOVL C01700 V=800.0 PL=0
MOVL C01701 V=800.0 PL=0
MOVL C01702 V=800.0 PL=0
MOVL C01703 V=800.0 PL=0
MOVL C01704 V=800.0 PL=0
MOVL C01705 V=800.0 PL=0
MOVL C01706 V=800.0 PL=0
MOVL C01707 V=800.0 PL=0
MOVL C01708 V=800.0 PL=0
MOVL C01709 V=800.0 PL=0
MOVL C01710 V=800.0 PL=0
MOVL C01711 V=800.0 PL=0
MOVL C01712 V=800.0 PL=0
MOVL C01713 V=800.0 PL=0
MOVL C01714 V=800.0 PL=0
MOVL C01715 V=800.0 PL=0
MOVL C01716 V=800.0 PL=0
MOVL C01717 V=800.0 PL=0
MOVL C01718 V=800.0 PL=0
MOVL C01719 V=800.0 PL=0
MOVL C01720 V=800.0 PL=0
MOVL C01721 V=800.0 PL=0
MOVL C01722 V=800.0 PL=0
MOVL C01723 V=800.0 PL=0
MOVL C01724 V=800.0 PL=0
MOVL C01725 V=800.0 PL=0
MOVL C01726 V=800.0 PL=0
MOVL C01727 V=800.0 PL=0
